C02371=1084,32291,-28357,1060,-27667,-1162
C02372=1082,32304,-28341,1060,-27672,-1161
C02373=1120,32308,-28336,1055,-27674,-1176
C02374=1156,32305,-28339,1050,-27673,-1190
C02375=1195,32311,-28332,1044,-27676,-1205
C02376=1230,32306,-28337,1039,-27674,-1219
C02377=1269,32312,-28330,1034,-27677,-1234
C02378=1304,32324,-28315,1028,-27682,-1248
C02379=1341,32332,-28305,1023,-27685,-1262
C02380=1378,32340,-28295,1018,-27689,-1277
C02381=1414,32352,-28280,1012,-27693,-1290
C02382=1452,32358,-28273,1007,-27696,-1305
C02383=1486,32373,-28255,1002,-27702,-1318
C02384=1521,32386,-28239,997,-27707,-1332
C02385=1556,32397,-28225,992,-27712,-1345
C02386=1592,32409,-28211,986,-27716,-1359
C02387=1624,32426,-28189,982,-27723,-1372
C02388=1655,32445,-28166,977,-27730,-1384
C02389=1688,32462,-28146,972,-27737,-1396
C02390=1718,32483,-28120,968,-27745,-1408
C02391=1749,32503,-28095,963,-27753,-1420
C02392=1781,32521,-28074,958,-27760,-1432
C02393=1810,32545,-28045,954,-27769,-1443
C02394=1838,32569,-28015,950,-27778,-1454
C02395=1867,32592,-27986,945,-27787,-1465
C02396=1892,32623,-27950,941,-27799,-1475
C02397=1921,32646,-27921,937,-27808,-1486
C02398=1946,32677,-27884,933,-27819,-1495
C02399=1971,32707,-27847,929,-27831,-1505
C02400=1996,32737,-27811,925,-27842,-1514
C02401=2022,32766,-27775,921,-27853,-1524
C02402=2018,32742,-27804,922,-27844,-1523
C02403=1993,32712,-27841,926,-27833,-1513
C02404=1975,32680,-27879,929,-27821,-1507
C02405=1950,32651,-27915,933,-27809,-1497
C02406=1921,32626,-27945,937,-27800,-1486
C02407=1896,32596,-27982,941,-27789,-1476
C02408=1867,32572,-28011,945,-27780,-1465
C02409=1839,32548,-28040,950,-27770,-1454
C02410=1810,32524,-28069,954,-27761,-1443
C02411=1781,32501,-28098,958,-27752,-1432
C02412=1752,32478,-28125,963,-27744,-1421
C02413=1718,32464,-28143,968,-27738,-1408
C02414=1688,32441,-28170,972,-27729,-1397
C02415=1655,32426,-28189,977,-27723,-1384
C02416=1621,32411,-28207,982,-27717,-1371
C02417=1589,32395,-28227,987,-27711,-1358
C02418=1554,32382,-28243,992,-27706,-1345
C02419=1520,32368,-28260,997,-27700,-1331
C02420=1486,32353,-28278,1002,-27695,-1318
C02421=1450,32343,-28291,1007,-27690,-1304
C02422=1413,32333,-28303,1013,-27686,-1290
C02423=1375,32328,-28310,1018,-27684,-1275
C02424=1341,32313,-28328,1023,-27678,-1262
C02425=1304,32304,-28340,1029,-27674,-1248
C02426=1268,32293,-28353,1034,-27670,-1234
C02427=1268,32293,-26953,1034,-27670,-1234
C02428=1269,32446,-24168,1032,-27726,-1233
C02429=1269,32446,-28168,1032,-27726,-1233
C02430=1230,32450,-28164,1037,-27727,-1218
C02431=1188,32444,-28172,1043,-27724,-1201
C02432=1149,32447,-28167,1049,-27726,-1186
C02433=1111,32451,-28163,1054,-27727,-1171
C02434=1072,32455,-28159,1060,-27728,-1156
C02435=1033,32459,-28154,1065,-27729,-1141
C02436=998,32473,-28138,1070,-27733,-1127
C02437=960,32477,-28133,1075,-27734,-1112
C02438=925,32491,-28117,1080,-27739,-1098
C02439=889,32503,-28103,1085,-27743,-1084
C02440=855,32519,-28084,1090,-27749,-1071
C02441=819,32530,-28070,1095,-27752,-1056
C02442=785,32547,-28050,1099,-27758,-1043
C02443=753,32571,-28022,1104,-27767,-1030
C02444=719,32589,-28001,1108,-27773,-1017
C02445=688,32613,-27972,1112,-27781,-1005
C02446=660,32639,-27940,1116,-27791,-994
C02447=632,32665,-27909,1119,-27800,-982
C02448=608,32693,-27876,1123,-27810,-973
C02449=590,32725,-26437,1125,-27821,-965
C02450=-41004,59868,4099,4900,-34257,16705
C02451=-41004,59868,1099,4900,-34257,16705
C02452=-41004,64596,1380,5213,-31659,16463
C02453=-41004,59868,1099,4900,-34257,16705
C02454=-41004,59868,9099,4900,-34257,16705
C02455=590,32725,-23837,1125,-27821,-965
C02456=590,32725,-27837,1125,-27821,-965
C02457=565,32753,-27804,1128,-27831,-955
C02458=553,32788,-27762,1129,-27844,-950
C02459=541,32823,-27720,1130,-27857,-945
C02460=540,32836,-27704,1130,-27862,-945
C02461=558,32804,-27742,1128,-27850,-952
C02462=576,32772,-27781,1126,-27839,-959
C02463=600,32744,-27814,1123,-27828,-969
C02464=618,32712,-27853,1121,-27817,-976
C02465=642,32684,-27886,1118,-27807,-986
C02466=674,32660,-27915,1114,-27798,-999
C02467=698,32632,-27949,1110,-27788,-1009
C02468=730,32608,-27978,1106,-27780,-1021
C02469=761,32583,-28007,1102,-27771,-1034
C02470=795,32566,-28027,1098,-27765,-1047
C02471=829,32549,-28047,1093,-27759,-1060
C02472=863,32532,-28068,1088,-27753,-1074
C02473=897,32516,-28087,1084,-27748,-1087
C02474=933,32505,-28100,1079,-27744,-1101
C02475=970,32495,-28112,1074,-27741,-1116
C02476=1006,32485,-28123,1069,-27738,-1130
C02477=1044,32480,-28129,1063,-27736,-1145
C02478=1082,32472,-28138,1058,-27734,-1160
C02479=1121,32469,-28141,1053,-27733,-1175
C02480=1159,32466,-28145,1047,-27733,-1190
C02481=1199,32464,-28147,1042,-27732,-1205
C02482=1240,32468,-28142,1036,-27734,-1221
C02483=1279,32466,-28143,1030,-27734,-1237
C02484=1321,32473,-28136,1024,-27737,-1253
C02485=1364,32479,-28128,1018,-27739,-1270
C02486=1401,32494,-28109,1013,-27745,-1284
C02487=1443,32500,-28102,1007,-27748,-1300
C02488=1478,32520,-28077,1001,-27756,-1314
C02489=1512,32537,-28056,996,-27763,-1327
C02490=1502,32518,-28079,998,-27755,-1323
C02491=1469,32494,-28108,1003,-27746,-1311
C02492=1432,32479,-28127,1008,-27740,-1296
C02493=1390,32473,-28134,1014,-27738,-1280
C02494=1351,32461,-28149,1020,-27733,-1265
C02495=1311,32452,-28161,1026,-27729,-1249
C02496=1269,32446,-28168,1032,-27726,-1233
C02497=1269,32446,-26768,1032,-27726,-1233
C02498=1271,32618,-23960,1029,-27790,-1232
C02499=1271,32618,-27960,1029,-27790,-1232
C02500=1216,32620,-27959,1037,-27790,-1211
C02501=1161,32621,-27958,1045,-27790,-1190
C02502=1110,32633,-27944,1052,-27793,-1169
C02503=1059,32644,-27930,1059,-27797,-1149
C02504=1009,32662,-27909,1066,-27803,-1130
C02505=963,32688,-27879,1072,-27812,-1111
C02506=915,32709,-27853,1079,-27819,-1092
C02507=871,32742,-27814,1085,-27831,-1075
C02508=827,32776,-27774,1090,-27843,-1058
C02509=790,32813,-27729,1095,-27856,-1043
C02510=756,32852,-27682,1099,-27870,-1029
C02511=724,32892,-27634,1103,-27885,-1016
C02512=700,32937,-27580,1106,-27901,-1007
C02513=670,32978,-27531,1110,-27916,-995
C02514=660,33023,-27477,1111,-27932,-990
C02515=689,32981,-27527,1107,-27917,-1002
C02516=719,32940,-27576,1103,-27902,-1014
C02517=749,32899,-27626,1100,-27887,-1026
C02518=785,32861,-27672,1095,-27874,-1040
C02519=816,32820,-27720,1091,-27859,-1053
C02520=853,32783,-27765,1087,-27846,-1068
C02521=897,32749,-27806,1081,-27834,-1085
C02522=943,32722,-27837,1075,-27825,-1103
C02523=989,32696,-27869,1069,-27815,-1122
C02524=1038,32676,-27892,1062,-27809,-1141
C02525=1087,32658,-27914,1055,-27802,-1160
C02526=1138,32646,-27927,1048,-27799,-1180
C02527=1193,32645,-27929,1040,-27799,-1202
C02528=1248,32643,-27930,1032,-27799,-1223
C02529=1303,32642,-27931,1025,-27799,-1245
C02530=1361,32650,-27920,1016,-27803,-1267
C02531=1420,32659,-27910,1008,-27807,-1290
C02532=1478,32668,-27899,1000,-27810,-1313
C02533=1532,32685,-27877,992,-27817,-1333
C02534=1586,32700,-27858,984,-27824,-1355
C02535=1639,32720,-27834,976,-27832,-1375
C02536=1692,32737,-27813,968,-27839,-1396
C02537=1741,32763,-27781,961,-27849,-1415
C02538=1789,32790,-27749,954,-27859,-1433
C02539=1838,32816,-27716,947,-27869,-1452
C02540=1879,32856,-27668,941,-27885,-1468
C02541=1921,32895,-27620,934,-27900,-1484
C02542=1962,32934,-27572,928,-27915,-1500
C02543=2000,32980,-27517,922,-27932,-1514
C02544=2009,32970,-27529,921,-27928,-1518
C02545=1978,32923,-27586,926,-27910,-1506
C02546=1939,32878,-27640,932,-27894,-1491
C02547=1899,32838,-27690,938,-27878,-1476
C02548=1857,32798,-27738,944,-27863,-1460
C02549=1809,32771,-27771,951,-27853,-1441
C02550=1759,32747,-27801,959,-27843,-1422
C02551=1711,32721,-27833,966,-27833,-1403
C02552=1661,32697,-27862,973,-27823,-1384
C02553=1608,32677,-27886,981,-27815,-1364
C02554=1554,32662,-27905,989,-27809,-1342
C02555=1496,32651,-27919,997,-27805,-1320
C02556=1438,32643,-27929,1006,-27801,-1297
C02557=1385,32625,-27951,1013,-27794,-1277
C02558=1326,32617,-27962,1022,-27790,-1254
C02559=1271,32618,-27960,1029,-27790,-1232
C02560=1271,32618,-26560,1029,-27790,-1232
C02561=998,32374,-24257,1071,-27697,-1128
C02562=998,32374,-28257,1071,-27697,-1128
C02563=1004,32369,-28263,1071,-27695,-1130
C02564=994,32367,-28265,1072,-27694,-1126
C02565=985,32366,-28267,1073,-27694,-1123
C02566=975,32365,-28269,1075,-27693,-1119
C02567=965,32363,-28271,1076,-27692,-1115
C02568=958,32369,-28264,1077,-27694,-1112
C02569=950,32371,-28262,1078,-27695,-1109
C02570=940,32369,-28264,1080,-27694,-1105
C02571=932,32371,-28261,1081,-27695,-1102
C02572=924,32376,-28255,1082,-27697,-1099
C02573=915,32375,-28257,1083,-27696,-1095
C02574=908,32381,-28250,1084,-27698,-1092
C02575=899,32382,-28248,1085,-27699,-1089
C02576=891,32385,-28245,1086,-27699,-1086
C02577=883,32389,-28240,1087,-27701,-1083
C02578=874,32389,-28241,1089,-27701,-1079
C02579=867,32394,-28234,1090,-27703,-1076
C02580=858,32395,-28233,1091,-27703,-1073
C02581=850,32398,-28230,1092,-27704,-1070
C02582=842,32403,-28224,1093,-27705,-1067
C02583=833,32402,-28225,1094,-27705,-1063
C02584=826,32408,-28218,1095,-27707,-1060
C02585=817,32408,-28217,1097,-27707,-1057
C02586=809,32411,-28214,1098,-27708,-1054
C02587=801,32416,-28209,1099,-27710,-1051
C02588=792,32415,-28209,1100,-27710,-1047
C02589=785,32421,-28202,1101,-27712,-1044
C02590=777,32427,-28196,1102,-27714,-1041
C02591=770,32432,-28189,1103,-27716,-1038
C02592=763,32438,-28183,1104,-27718,-1036
C02593=761,32446,-28172,1104,-27721,-1035
C02594=767,32444,-28175,1103,-27720,-1037
C02595=775,32440,-28179,1102,-27719,-1040
C02596=784,32440,-28180,1101,-27718,-1044
C02597=791,32434,-28187,1100,-27717,-1047
C02598=798,32429,-28193,1099,-27715,-1049
C02599=806,32426,-28196,1098,-27714,-1053
C02600=815,32425,-28198,1097,-27713,-1056
C02601=822,32419,-28204,1096,-27711,-1059
C02602=832,32420,-28203,1094,-27712,-1063
C02603=839,32415,-28209,1093,-27710,-1065
C02604=848,32413,-28212,1092,-27709,-1069
C02605=856,32411,-28214,1091,-27709,-1072
C02606=863,32406,-28220,1090,-27707,-1075
C02607=870,32400,-28227,1089,-27705,-1078
C02608=879,32398,-28229,1088,-27704,-1081
C02609=889,32400,-28227,1087,-27705,-1085
C02610=897,32398,-28230,1085,-27704,-1088
C02611=904,32393,-28236,1084,-27702,-1091
C02612=914,32394,-28234,1083,-27703,-1095
C02613=921,32388,-28241,1082,-27701,-1098
C02614=930,32387,-28243,1081,-27701,-1101
C02615=938,32384,-28245,1080,-27700,-1104
C02616=945,32379,-28251,1079,-27698,-1107
C02617=955,32381,-28249,1077,-27699,-1111
C02618=965,32382,-28248,1076,-27699,-1115
C02619=972,32376,-28255,1075,-27697,-1118
C02620=980,32375,-28256,1074,-27697,-1121
C02621=990,32376,-28255,1072,-27698,-1125
C02622=998,32374,-26857,1071,-27697,-1128
C02623=-41004,59868,4099,4900,-34257,16705
C02624=-41004,59868,1099,4900,-34257,16705
C02625=-41004,64596,1380,5213,-31659,16463
C02626=-41004,59868,1099,4900,-34257,16705
C02627=-41004,59868,9099,4900,-34257,16705
C02628=998,32374,-24257,1071,-27697,-1128
C02629=998,32374,-28257,1071,-27697,-1128
C02630=998,32374,-26857,1071,-27697,-1128
C02631=975,32976,-23531,1067,-27918,-1114
C02632=975,32976,-27531,1067,-27918,-1114
C02633=961,32984,-27522,1069,-27921,-1108
C02634=947,32989,-27515,1071,-27923,-1103
C02635=934,32999,-27503,1072,-27926,-1097
C02636=921,33009,-27491,1074,-27930,-1092
C02637=913,33022,-27476,1075,-27935,-1089
C02638=902,33033,-27463,1077,-27939,-1085
C02639=889,33043,-27451,1078,-27942,-1079
C02640=881,33056,-27435,1079,-27947,-1076
C02641=871,33067,-27422,1081,-27951,-1072
C02642=864,33080,-27406,1081,-27956,-1069
C02643=857,33094,-27389,1082,-27961,-1067
C02644=848,33106,-27374,1083,-27965,-1063
C02645=838,33118,-27361,1084,-27969,-1059
C02646=832,33132,-27344,1085,-27974,-1056
C02647=826,33146,-27327,1086,-27979,-1054
C02648=816,33157,-27314,1087,-27983,-1050
C02649=807,33169,-27299,1088,-27988,-1046
C02650=804,33185,-27280,1088,-27994,-1045
C02651=795,33197,-27266,1090,-27998,-1041
C02652=793,33213,-27246,1090,-28004,-1040
C02653=789,33228,-27228,1090,-28009,-1039
C02654=781,33241,-27213,1091,-28014,-1036
C02655=780,33258,-27192,1091,-28020,-1035
C02656=779,33275,-27172,1091,-28026,-1034
C02657=771,33287,-27157,1092,-28031,-1031
C02658=767,33303,-27139,1092,-28036,-1030
C02659=766,33319,-27118,1092,-28042,-1029
C02660=765,33336,-27098,1092,-28049,-1029
C02661=764,33353,-27078,1092,-28055,-1028
C02662=766,33363,-27066,1091,-28059,-1029
C02663=774,33350,-27081,1090,-28054,-1032
C02664=775,33333,-27101,1091,-28048,-1032
C02665=776,33317,-27121,1091,-28042,-1033
C02666=784,33304,-27137,1090,-28037,-1036
C02667=788,33289,-27155,1089,-28032,-1038
C02668=789,33272,-27175,1089,-28025,-1038
C02669=790,33255,-27195,1089,-28019,-1039
C02670=800,33244,-27209,1088,-28015,-1043
C02671=802,33227,-27229,1088,-28009,-1044
C02672=808,33214,-27245,1088,-28004,-1046
C02673=813,33199,-27263,1087,-27999,-1048
C02674=820,33186,-27279,1086,-27994,-1051
C02675=825,33171,-27296,1086,-27989,-1053
C02676=833,33158,-27312,1085,-27984,-1056
C02677=839,33145,-27328,1084,-27979,-1059
C02678=847,33132,-27344,1083,-27974,-1062
C02679=857,33121,-27357,1082,-27970,-1066
C02680=864,33107,-27374,1081,-27965,-1069
C02681=870,33093,-27390,1080,-27960,-1072
C02682=880,33081,-27405,1079,-27956,-1075
C02683=889,33069,-27419,1078,-27952,-1079
C02684=901,33059,-27432,1076,-27948,-1084
C02685=908,33046,-27447,1075,-27943,-1087
C02686=921,33036,-27459,1074,-27940,-1092
C02687=933,33025,-27472,1072,-27936,-1097
C02688=940,33012,-27488,1071,-27931,-1100
C02689=953,33002,-27500,1070,-27928,-1105
C02690=966,32992,-27512,1068,-27924,-1110
C02691=979,32982,-27524,1066,-27921,-1115
C02692=975,32976,-27531,1067,-27918,-1114
C02693=975,32976,-26131,1067,-27918,-1114
C02694=1115,33029,-23465,1046,-27940,-1168
C02695=1115,33029,-27465,1046,-27940,-1168
C02696=1109,33039,-27453,1047,-27943,-1166
C02697=1102,33049,-27442,1048,-27947,-1163
C02698=1092,33057,-27432,1050,-27950,-1159
C02699=1087,33068,-27419,1050,-27954,-1157
C02700=1078,33076,-27409,1051,-27957,-1153
C02701=1074,33088,-27395,1052,-27961,-1152
C02702=1066,33097,-27384,1053,-27964,-1148
C02703=1061,33108,-27371,1053,-27968,-1146
C02704=1054,33118,-27359,1054,-27972,-1144
C02705=1047,33127,-27348,1055,-27975,-1140
C02706=1043,33139,-27334,1055,-27979,-1139
C02707=1033,33147,-27324,1057,-27982,-1135
C02708=1032,33160,-27308,1057,-27987,-1134
C02709=1026,33170,-27296,1057,-27991,-1132
C02710=1021,33181,-27283,1058,-27995,-1130
C02711=1029,33177,-27288,1057,-27993,-1133
C02712=1039,33169,-27297,1056,-27990,-1137
C02713=1043,33157,-27311,1055,-27986,-1139
C02714=1052,33149,-27321,1054,-27983,-1142
C02715=1056,33138,-27335,1053,-27979,-1144
C02716=1064,33128,-27346,1053,-27976,-1147
C02717=1070,33118,-27358,1052,-27972,-1150
C02718=1075,33107,-27371,1051,-27968,-1152
C02719=1084,33099,-27382,1050,-27965,-1155
C02720=1087,33087,-27396,1050,-27961,-1157
C02721=1097,33079,-27406,1049,-27958,-1160
C02722=1101,33067,-27419,1048,-27954,-1162
C02723=1111,33059,-27429,1047,-27951,-1166
C02724=1121,33052,-27438,1045,-27948,-1170
C02725=1132,33044,-27448,1044,-27945,-1174
C02726=1142,33036,-27457,1043,-27943,-1178
C02727=1152,33028,-27467,1041,-27940,-1182
C02728=1163,33023,-27473,1040,-27938,-1187
C02729=1175,33019,-27477,1038,-27937,-1191
C02730=1187,33017,-27480,1037,-27936,-1196
C02731=1198,33010,-27487,1035,-27934,-1201
C02732=1211,33010,-27488,1033,-27934,-1205
C02733=1221,33003,-27496,1032,-27931,-1210
C02734=1235,33005,-27494,1030,-27932,-1215
C02735=1246,33000,-27499,1028,-27931,-1219
C02736=1259,32999,-27501,1027,-27930,-1224
C02737=1272,32999,-27501,1025,-27930,-1229
C02738=1282,32992,-27508,1023,-27928,-1234
C02739=1294,32990,-27511,1022,-27927,-1238
C02740=1294,32985,-27517,1022,-27925,-1238
C02741=1281,32983,-27520,1024,-27925,-1233
C02742=1270,32991,-27511,1025,-27927,-1229
C02743=1257,32989,-27513,1027,-27926,-1224
C02744=1245,32992,-27509,1029,-27928,-1219
C02745=1233,32995,-27506,1030,-27928,-1214
C02746=1220,32994,-27507,1032,-27928,-1209
C02747=1209,33001,-27499,1034,-27930,-1205
C02748=1196,32999,-27501,1036,-27930,-1200
C02749=1184,33003,-27496,1037,-27931,-1195
C02750=1172,33005,-27494,1039,-27931,-1190
C02751=1161,33012,-27486,1040,-27934,-1186
C02752=1149,33013,-27485,1042,-27934,-1181
C02753=1138,33019,-27477,1043,-27936,-1177
C02754=1126,33021,-27475,1045,-27937,-1172
C02755=1115,33029,-27465,1046,-27940,-1168
C02756=1115,33029,-26065,1046,-27940,-1168
C02757=1159,33118,-23358,1039,-27973,-1185
C02758=1159,33118,-27358,1039,-27973,-1185
C02759=1098,33196,-27264,1047,-28001,-1160
C02760=1121,33177,-27286,1044,-27995,-1169
C02761=1204,33114,-27363,1033,-27972,-1202
C02762=1299,33071,-27413,1020,-27957,-1239
C02763=1397,33036,-27454,1007,-27946,-1278
C02764=1499,33015,-27479,992,-27939,-1318
C02765=1611,33022,-27470,977,-27943,-1362
C02766=1719,33039,-27448,961,-27951,-1404
C02767=1667,33068,-27414,968,-27961,-1383
C02768=1559,33073,-27408,983,-27961,-1341
C02769=1460,33104,-27371,997,-27972,-1302
C02770=1365,33150,-27317,1010,-27987,-1265
C02771=1278,33217,-27237,1021,-28011,-1230
C02772=1200,33289,-27151,1031,-28037,-1199
C02773=1136,33369,-27055,1039,-28065,-1173
C02774=1085,33456,-26950,1045,-28097,-1153
C02775=1055,33555,-26831,1049,-28133,-1140
C02776=1038,33661,-26703,1050,-28172,-1132
C02777=1048,33768,-26573,1047,-28212,-1136
C02778=1081,33870,-26451,1041,-28250,-1148
C02779=1142,33964,-26336,1031,-28285,-1171
C02780=1176,33974,-26324,1027,-28289,-1184
C02781=1101,33883,-26435,1038,-28255,-1155
C02782=1069,33781,-26558,1044,-28217,-1144
C02783=1066,33672,-26690,1045,-28176,-1144
C02784=1083,33565,-26818,1044,-28137,-1151
C02785=1110,33465,-26940,1042,-28100,-1162
C02786=1162,33378,-27043,1036,-28069,-1184
C02787=1229,33300,-27137,1027,-28041,-1210
C02788=1303,33226,-27226,1018,-28015,-1240
C02789=1392,33166,-27298,1006,-27993,-1275
C02790=1485,33118,-27355,993,-27977,-1312
C02791=1585,33088,-27390,979,-27967,-1351
C02792=1693,33081,-27397,964,-27966,-1393
C02793=1800,33112,-27359,949,-27978,-1435
C02794=1758,33139,-27327,955,-27988,-1418
C02795=1697,33139,-27327,963,-27987,-1395
C02796=1631,33177,-27282,972,-28001,-1368
C02797=1529,33201,-27254,986,-28008,-1328
C02798=1435,33248,-25798,999,-28024,-1291
C02799=-41004,59868,4099,4900,-34257,16705
C02800=-41004,59868,1099,4900,-34257,16705
C02801=-41004,64596,1380,5213,-31659,16463
C02802=-41004,59868,1099,4900,-34257,16705
C02803=-41004,59868,9099,4900,-34257,16705
C02804=1435,33248,-23198,999,-28024,-1291
C02805=1435,33248,-27198,999,-28024,-1291
C02806=1355,33319,-27113,1009,-28050,-1259
C02807=1282,33393,-27024,1019,-28076,-1230
C02808=1235,33483,-26916,1024,-28109,-1211
C02809=1200,33579,-26800,1028,-28144,-1197
C02810=1245,33495,-26902,1023,-28113,-1215
C02811=1297,33408,-27006,1016,-28082,-1236
C02812=1370,33334,-27095,1007,-28055,-1265
C02813=1451,33263,-27180,996,-28030,-1297
C02814=1543,33212,-27240,984,-28012,-1334
C02815=1644,33186,-27271,970,-28004,-1373
C02816=1748,33169,-27291,956,-27999,-1414
C02817=1861,33185,-27270,939,-28006,-1458
C02818=1858,33129,-27338,941,-27985,-1457
C02819=1769,33063,-27418,954,-27960,-1423
C02820=1667,33020,-27471,969,-27943,-1384
C02821=1557,32994,-27503,985,-27932,-1341
C02822=1448,32998,-27500,1000,-27932,-1298
C02823=1349,33029,-27464,1014,-27942,-1259
C02824=1252,33067,-27418,1027,-27956,-1221
C02825=1159,33118,-27358,1039,-27973,-1185
C02826=1159,33118,-25958,1039,-27973,-1185
C02827=964,33299,-23141,1064,-28038,-1107
C02828=964,33299,-27141,1064,-28038,-1107
C02829=953,33311,-27126,1066,-28042,-1102
C02830=943,33324,-27111,1067,-28046,-1098
C02831=936,33338,-27094,1068,-28052,-1095
C02832=930,33353,-27076,1069,-28057,-1093
C02833=920,33366,-27061,1070,-28062,-1089
C02834=916,33381,-27042,1070,-28067,-1087
C02835=908,33396,-27025,1071,-28072,-1084
C02836=907,33413,-27004,1071,-28079,-1083
C02837=906,33431,-26983,1071,-28085,-1083
C02838=905,33448,-26961,1071,-28092,-1082
C02839=895,33461,-26946,1072,-28096,-1078
C02840=893,33478,-26925,1072,-28103,-1077
C02841=892,33496,-26904,1072,-28109,-1077
C02842=891,33513,-26883,1072,-28116,-1076
C02843=890,33531,-26862,1072,-28122,-1076
C02844=889,33548,-26841,1072,-28129,-1075
C02845=888,33566,-26819,1072,-28135,-1074
C02846=887,33584,-26798,1072,-28141,-1074
C02847=885,33601,-26777,1072,-28148,-1073
C02848=884,33619,-26756,1072,-28154,-1073
C02849=887,33635,-26736,1071,-28161,-1074
C02850=892,33651,-26716,1070,-28167,-1075
C02851=891,33669,-26695,1070,-28173,-1075
C02852=890,33687,-26674,1070,-28179,-1074
C02853=892,33703,-26654,1069,-28186,-1075
C02854=897,33719,-26634,1069,-28192,-1077
C02855=896,33737,-26613,1069,-28198,-1076
C02856=900,33753,-26593,1068,-28204,-1078
C02857=904,33769,-26574,1067,-28210,-1079
C02858=913,33779,-26562,1066,-28214,-1082
C02859=923,33767,-26577,1064,-28210,-1087
C02860=915,33751,-26595,1066,-28204,-1084
C02861=916,33734,-26616,1066,-28197,-1084
C02862=913,33718,-26636,1066,-28191,-1083
C02863=908,33701,-26656,1067,-28185,-1081
C02864=909,33684,-26677,1067,-28179,-1082
C02865=910,33666,-26698,1067,-28172,-1083
C02866=912,33649,-26719,1067,-28166,-1083
C02867=909,33632,-26740,1068,-28160,-1082
C02868=904,33616,-26759,1069,-28154,-1080
C02869=905,33598,-26780,1069,-28147,-1081
C02870=906,33581,-26801,1069,-28141,-1082
C02871=907,33563,-26822,1069,-28134,-1082
C02872=909,33546,-26844,1069,-28128,-1083
C02873=910,33528,-26865,1069,-28121,-1083
C02874=911,33511,-26886,1069,-28115,-1084
C02875=912,33493,-26907,1069,-28108,-1085
C02876=913,33475,-26928,1069,-28102,-1085
C02877=914,33458,-26950,1069,-28095,-1086
C02878=915,33440,-26971,1070,-28089,-1086
C02879=926,33428,-26986,1068,-28085,-1090
C02880=927,33410,-27007,1068,-28078,-1091
C02881=928,33393,-27028,1068,-28072,-1092
C02882=939,33381,-27043,1067,-28067,-1096
C02883=940,33363,-27064,1067,-28061,-1097
C02884=951,33351,-27079,1066,-28056,-1101
C02885=953,33334,-27099,1066,-28050,-1102
C02886=962,33321,-27114,1064,-28046,-1106
C02887=973,33309,-27129,1063,-28041,-1110
C02888=964,33299,-27141,1064,-28038,-1107
C02889=964,33299,-25741,1064,-28038,-1107
C02890=523,33294,-23151,1127,-28030,-934
C02891=523,33294,-27151,1127,-28030,-934
C02892=524,33274,-27175,1127,-28023,-935
C02893=525,33254,-27200,1127,-28015,-935
C02894=526,33233,-27224,1127,-28008,-936
C02895=536,33218,-27243,1126,-28002,-940
C02896=538,33198,-27267,1126,-27995,-941
C02897=539,33178,-27291,1126,-27988,-942
C02898=541,33158,-27316,1126,-27980,-942
C02899=545,33139,-27338,1125,-27973,-944
C02900=553,33122,-27358,1125,-27967,-947
C02901=554,33102,-27382,1125,-27960,-948
C02902=564,33087,-27400,1123,-27955,-952
C02903=567,33068,-27424,1123,-27947,-953
C02904=576,33052,-27443,1122,-27942,-957
C02905=585,33036,-27462,1121,-27936,-961
C02906=588,33017,-27485,1121,-27929,-962
C02907=599,33002,-27503,1120,-27923,-966
C02908=610,32987,-27521,1118,-27918,-971
C02909=611,32967,-27545,1118,-27911,-971
C02910=622,32952,-27563,1117,-27905,-976
C02911=632,32936,-27582,1116,-27900,-980
C02912=613,32933,-27587,1119,-27898,-973
C02913=611,32952,-27563,1119,-27905,-972
C02914=601,32968,-27544,1120,-27911,-968
C02915=590,32983,-27526,1121,-27916,-963
C02916=584,33000,-27505,1122,-27923,-961
C02917=575,33016,-27486,1123,-27928,-957
C02918=568,33033,-27466,1124,-27935,-954
C02919=557,33048,-27448,1125,-27940,-950
C02920=555,33068,-27424,1125,-27947,-949
C02921=545,33083,-27406,1126,-27953,-945
C02922=538,33100,-27386,1127,-27959,-942
C02923=533,33118,-27363,1127,-27966,-940
C02924=532,33138,-27339,1127,-27973,-939
C02925=524,33155,-27319,1128,-27979,-936
C02926=520,33174,-27296,1129,-27986,-934
C02927=519,33194,-27272,1128,-27993,-933
C02928=518,33214,-27248,1128,-28001,-933
C02929=516,33235,-27223,1128,-28008,-932
C02930=507,33250,-27204,1129,-28014,-928
C02931=505,33270,-27181,1129,-28021,-927
C02932=503,33290,-27156,1129,-28028,-926
C02933=502,33310,-27132,1129,-28036,-926
C02934=501,33331,-27107,1129,-28043,-925
C02935=510,33348,-27086,1128,-28050,-928
C02936=509,33369,-27061,1128,-28058,-928
C02937=507,33389,-27037,1127,-28065,-927
C02938=506,33409,-27012,1127,-28072,-926
C02939=510,33428,-26989,1127,-28080,-928
C02940=514,33447,-26966,1126,-28087,-929
C02941=513,33468,-26942,1126,-28094,-928
C02942=527,33469,-26940,1124,-28095,-934
C02943=523,33454,-26958,1124,-28089,-933
C02944=524,33434,-26983,1124,-28082,-933
C02945=525,33413,-27007,1125,-28074,-934
C02946=524,33394,-27031,1125,-28067,-933
C02947=518,33375,-27053,1126,-28060,-931
C02948=519,33355,-27078,1126,-28053,-932
C02949=520,33335,-27102,1126,-28045,-933
C02950=522,33315,-27126,1126,-28038,-933
C02951=523,33294,-27151,1127,-28030,-934
C02952=523,33294,-25751,1127,-28030,-934
C02953=303,33334,-23105,1157,-28042,-848
C02954=303,33334,-27105,1157,-28042,-848
C02955=303,33367,-27065,1156,-28054,-847
C02956=311,33398,-27027,1155,-28066,-850
C02957=309,33432,-26987,1155,-28078,-849
C02958=317,33463,-26949,1153,-28090,-852
C02959=325,33494,-26911,1152,-28101,-855
C02960=333,33525,-26874,1150,-28113,-858
C02961=341,33557,-26836,1148,-28125,-861
C02962=349,33588,-26799,1147,-28136,-863
C02963=363,33617,-26763,1145,-28147,-868
C02964=379,33647,-26727,1142,-28158,-874
C02965=395,33676,-26692,1139,-28169,-880
C02966=418,33703,-26659,1136,-28180,-889
C02967=433,33732,-26623,1133,-28190,-895
C02968=460,33753,-26598,1129,-28199,-905
C02969=482,33781,-26564,1126,-28209,-914
C02970=508,33802,-26539,1122,-28217,-924
C02971=536,33819,-26517,1118,-28224,-935
C02972=561,33842,-26490,1114,-28233,-944
C02973=591,33856,-26473,1110,-28238,-956
C02974=601,33880,-25043,1108,-28247,-959
C02975=-41004,59868,4099,4900,-34257,16705
C02976=-41004,59868,1099,4900,-34257,16705
C02977=-41004,64596,1380,5213,-31659,16463
C02978=-41004,59868,1099,4900,-34257,16705
C02979=-41004,59868,9099,4900,-34257,16705
C02980=601,33880,-22443,1108,-28247,-959
C02981=601,33880,-26443,1108,-28247,-959
C02982=573,33893,-26427,1112,-28252,-948
C02983=545,33906,-26412,1115,-28256,-937
C02984=517,33920,-26396,1119,-28261,-926
C02985=491,33940,-26372,1122,-28268,-916
C02986=463,33953,-26357,1126,-28272,-905
C02987=438,33973,-26333,1129,-28279,-895
C02988=410,33986,-26317,1133,-28284,-883
C02989=384,34006,-26293,1136,-28291,-873
C02990=359,34027,-26269,1140,-28298,-863
C02991=333,34047,-26245,1143,-28305,-853
C02992=314,34071,-26216,1145,-28314,-845
C02993=292,34093,-26190,1148,-28321,-836
C02994=271,34116,-26162,1151,-28330,-828
C02995=251,34139,-26134,1153,-28338,-820
C02996=232,34131,-26144,1156,-28335,-812
C02997=233,34098,-26184,1156,-28322,-813
C02998=245,34070,-26218,1155,-28312,-818
C02999=247,34036,-26259,1155,-28300,-819
C03000=248,34002,-26299,1155,-28287,-820
C03001=250,33969,-26340,1156,-28275,-821
C03002=252,33935,-26381,1156,-28263,-822
C03003=254,33901,-26421,1156,-28250,-823
C03004=256,33868,-26462,1156,-28238,-824
C03005=258,33834,-26502,1156,-28226,-825
C03006=260,33800,-26543,1157,-28213,-826
C03007=261,33767,-26583,1157,-28201,-827
C03008=263,33733,-26624,1157,-28189,-828
C03009=265,33699,-26665,1157,-28176,-829
C03010=267,33666,-26705,1157,-28164,-830
C03011=269,33632,-26746,1158,-28152,-832
C03012=271,33599,-26786,1158,-28139,-833
C03013=273,33565,-26827,1158,-28127,-834
C03014=275,33531,-26867,1158,-28114,-835
C03015=276,33498,-26908,1158,-28102,-836
C03016=270,33466,-26946,1160,-28090,-833
C03017=270,33433,-26986,1160,-28078,-834
C03018=272,33399,-27027,1160,-28066,-835
C03019=274,33366,-27067,1160,-28053,-836
C03020=276,33332,-27108,1161,-28041,-837
C03021=303,33334,-27105,1157,-28042,-848
C03022=303,33334,-25705,1157,-28042,-848
C03023=1429,33520,-22870,996,-28125,-1287
C03024=1429,33520,-26870,996,-28125,-1287
C03025=1428,33538,-26848,996,-28131,-1286
C03026=1417,33551,-26832,998,-28136,-1282
C03027=1416,33569,-26811,998,-28143,-1281
C03028=1407,33583,-26794,999,-28148,-1277
C03029=1404,33600,-26773,999,-28154,-1276
C03030=1403,33618,-26751,999,-28161,-1276
C03031=1401,33636,-26729,999,-28167,-1275
C03032=1400,33655,-26707,999,-28174,-1274
C03033=1402,33667,-26693,999,-28179,-1275
C03034=1410,33652,-26710,998,-28173,-1278
C03035=1411,33634,-26732,998,-28167,-1279
C03036=1418,33619,-26751,997,-28161,-1281
C03037=1423,33603,-26770,996,-28155,-1284
C03038=1425,33585,-26791,996,-28149,-1284
C03039=1433,33571,-26808,995,-28144,-1288
C03040=1437,33554,-26829,995,-28137,-1289
C03041=1447,33541,-26844,994,-28133,-1294
C03042=1449,33523,-26866,994,-28126,-1294
C03043=1457,33508,-26884,993,-28121,-1298
C03044=1461,33492,-26904,992,-28115,-1299
C03045=1472,33479,-26919,991,-28110,-1304
C03046=1479,33464,-26937,990,-28105,-1307
C03047=1484,33448,-26956,990,-28099,-1309
C03048=1494,33435,-26972,988,-28094,-1313
C03049=1502,33420,-26990,987,-28089,-1316
C03050=1509,33405,-27007,987,-28083,-1319
C03051=1517,33391,-27025,986,-28078,-1322
C03052=1528,33378,-27040,984,-28074,-1327
C03053=1538,33365,-27056,983,-28069,-1331
C03054=1546,33350,-27073,982,-28064,-1334
C03055=1553,33336,-27091,981,-28058,-1337
C03056=1568,33325,-27104,979,-28054,-1342
C03057=1575,33310,-27122,978,-28049,-1346
C03058=1589,33299,-27135,976,-28045,-1351
C03059=1603,33288,-27148,975,-28041,-1357
C03060=1611,33274,-27166,974,-28036,-1360
C03061=1625,33263,-27179,972,-28032,-1365
C03062=1639,33252,-27192,970,-28028,-1371
C03063=1637,33245,-27200,970,-28026,-1370
C03064=1621,33252,-27191,973,-28028,-1364
C03065=1606,33260,-27182,975,-28031,-1358
C03066=1591,33271,-27169,976,-28035,-1352
C03067=1577,33282,-27156,978,-28038,-1347
C03068=1570,33296,-27139,979,-28044,-1344
C03069=1556,33307,-27125,981,-28048,-1338
C03070=1548,33322,-27108,982,-28053,-1335
C03071=1534,33333,-27095,984,-28057,-1329
C03072=1526,33348,-27077,985,-28062,-1326
C03073=1512,33358,-27064,987,-28066,-1321
C03074=1505,33373,-27046,988,-28071,-1317
C03075=1497,33388,-27029,988,-28077,-1314
C03076=1487,33401,-27013,990,-28082,-1310
C03077=1482,33417,-26993,990,-28087,-1308
C03078=1475,33432,-26976,991,-28093,-1305
C03079=1464,33445,-26960,992,-28097,-1301
C03080=1453,33458,-26945,994,-28102,-1297
C03081=1452,33476,-26923,994,-28109,-1296
C03082=1441,33489,-26907,995,-28113,-1292
C03083=1437,33505,-26887,995,-28119,-1290
C03084=1429,33520,-26870,996,-28125,-1287
C03085=1429,33520,-25470,996,-28125,-1287
C03086=1682,33546,-22836,961,-28138,-1386
C03087=1682,33546,-26836,961,-28138,-1386
C03088=1695,33511,-26879,959,-28125,-1391
C03089=1708,33475,-26921,958,-28112,-1396
C03090=1729,33445,-26958,955,-28101,-1405
C03091=1751,33415,-26994,952,-28090,-1414
C03092=1774,33384,-27030,950,-28079,-1423
C03093=1796,33354,-27066,947,-28068,-1431
C03094=1821,33326,-27100,944,-28058,-1442
C03095=1855,33306,-27125,939,-28051,-1455
C03096=1890,33291,-27142,934,-28046,-1469
C03097=1924,33274,-27163,930,-28040,-1482
C03098=1961,33263,-27175,924,-28036,-1497
C03099=2000,33260,-27178,919,-28036,-1512
C03100=2039,33256,-27183,914,-28035,-1527
C03101=2076,33271,-27164,908,-28041,-1542
C03102=2115,33268,-27168,903,-28040,-1557
C03103=2144,33292,-27138,898,-28049,-1568
C03104=2111,33315,-27111,903,-28057,-1555
C03105=2072,33319,-27107,908,-28058,-1540
C03106=2033,33322,-27103,914,-28059,-1525
C03107=1997,33334,-27089,919,-28063,-1510
C03108=1962,33350,-27070,923,-28068,-1497
C03109=1928,33369,-27048,928,-28075,-1483
C03110=1901,33396,-27015,932,-28085,-1472
C03111=1877,33425,-26980,935,-28095,-1463
C03112=1856,33456,-26943,937,-28106,-1454
C03113=1834,33486,-26907,940,-28117,-1446
C03114=1814,33518,-26869,942,-28129,-1438
C03115=1800,33552,-26827,944,-28141,-1432
C03116=1787,33588,-26785,945,-28154,-1426
C03117=1775,33623,-26742,947,-28167,-1421
C03118=1771,33664,-26692,947,-28182,-1420
C03119=1759,33699,-26650,948,-28195,-1414
C03120=1756,33740,-26600,948,-28210,-1413
C03121=1762,33779,-26554,947,-28225,-1415
C03122=1769,33817,-26507,945,-28239,-1418
C03123=1781,33854,-26462,943,-28253,-1422
C03124=1794,33891,-26418,941,-28267,-1427
C03125=1819,33925,-26377,937,-28279,-1436
C03126=1844,33954,-26341,933,-28291,-1446
C03127=1877,33978,-26312,929,-28300,-1458
C03128=1913,33994,-26292,923,-28306,-1472
C03129=1934,34020,-26261,920,-28316,-1480
C03130=1900,34037,-26240,925,-28322,-1467
C03131=1863,34048,-26228,930,-28325,-1453
C03132=1827,34058,-26215,935,-28329,-1438
C03133=1795,34047,-26229,939,-28324,-1426
C03134=1761,34027,-26254,944,-28316,-1413
C03135=1731,34000,-26287,949,-28306,-1401
C03136=1703,33967,-26327,953,-28293,-1391
C03137=1683,33931,-26370,956,-28280,-1383
C03138=1675,33893,-26416,958,-28266,-1380
C03139=1664,33856,-26461,960,-28252,-1376
C03140=1652,33819,-26506,962,-28238,-1372
C03141=1651,33779,-26554,962,-28223,-1372
C03142=1648,33740,-26602,963,-28209,-1371
C03143=1651,33699,-26651,963,-28194,-1372
C03144=1655,33658,-26700,963,-28179,-1374
C03145=1667,33623,-26743,962,-28166,-1379
C03146=1670,33582,-26793,962,-28151,-1380
C03147=1682,33546,-25436,961,-28138,-1386
C03148=-41004,59868,4099,4900,-34257,16705
C03149=-41004,59868,1099,4900,-34257,16705
C03150=-41004,64596,1380,5213,-31659,16463
C03151=-41004,59868,1099,4900,-34257,16705
C03152=-41004,59868,9099,4900,-34257,16705
C03153=1682,33546,-22836,961,-28138,-1386
C03154=1682,33546,-26836,961,-28138,-1386
C03155=1682,33546,-25436,961,-28138,-1386
C03156=1856,33512,-22875,937,-28127,-1454
C03157=1856,33512,-26875,937,-28127,-1454
C03158=1974,33377,-27037,921,-28079,-1501
C03159=2151,33340,-27081,897,-28067,-1571
C03160=2340,33372,-27041,870,-28081,-1644
C03161=2512,33450,-26944,845,-28112,-1711
C03162=2684,33529,-26847,820,-28143,-1777
C03163=2856,33605,-26754,795,-28174,-1844
C03164=3022,33693,-26646,770,-28208,-1909
C03165=3169,33814,-26497,749,-28255,-1965
C03166=3326,33900,-26392,726,-28289,-2026
C03167=3484,34001,-26269,703,-28328,-2087
C03168=3644,34095,-26153,679,-28365,-2149
C03169=3479,34101,-26148,703,-28365,-2085
C03170=3332,33982,-26293,724,-28319,-2028
C03171=3201,33903,-26389,743,-28289,-1977
C03172=3344,34029,-26236,722,-28337,-2033
C03173=3484,34160,-26075,701,-28388,-2086
C03174=3612,34311,-25892,682,-28445,-2136
C03175=3723,34470,-25698,665,-28506,-2178
C03176=3825,34622,-25513,650,-28564,-2217
C03177=3689,34665,-25463,669,-28578,-2164
C03178=3555,34527,-25631,689,-28525,-2112
C03179=3420,34389,-25799,709,-28472,-2060
C03180=3274,34270,-25945,730,-28426,-2004
C03181=3121,34161,-26078,752,-28383,-1944
C03182=3199,34325,-25878,740,-28445,-1974
C03183=3331,34470,-25703,720,-28501,-2025
C03184=3462,34614,-25527,701,-28556,-2075
C03185=3576,34767,-25339,684,-28615,-2119
C03186=3671,34931,-25140,669,-28677,-2155
C03187=3638,35070,-24972,673,-28728,-2142
C03188=3490,34958,-25109,694,-28684,-2084
C03189=3352,34827,-25270,714,-28634,-2031
C03190=3218,34689,-25438,734,-28581,-1979
C03191=3086,34545,-25614,754,-28525,-1928
C03192=2957,34394,-25797,773,-28468,-1879
C03193=2973,34446,-25735,771,-28487,-1885
C03194=3100,34598,-25549,751,-28545,-1934
C03195=3232,34742,-25374,732,-28601,-1985
C03196=3368,34878,-25208,712,-28653,-2037
C03197=3478,35008,-25049,695,-28703,-2080
C03198=3306,35030,-25024,719,-28709,-2012
C03199=3156,34922,-25157,741,-28667,-1953
C03200=3005,34814,-25289,763,-28624,-1895
C03201=2869,34676,-25458,783,-28571,-1843
C03202=2735,34535,-25630,803,-28517,-1791
C03203=2834,34674,-25461,788,-28570,-1829
C03204=2966,34818,-25285,768,-28625,-1880
C03205=3117,34926,-25152,746,-28667,-1938
C03206=3047,34992,-25073,755,-28691,-1910
C03207=2876,34919,-25163,780,-28662,-1844
C03208=2720,34820,-25285,802,-28623,-1783
C03209=2596,34672,-25466,821,-28566,-1736
C03210=2467,34521,-25649,840,-28509,-1686
C03211=2334,34377,-25825,860,-28453,-1635
C03212=2214,34218,-26018,879,-28393,-1589
C03213=2114,34054,-26217,894,-28331,-1551
C03214=1957,33990,-26297,917,-28305,-1490
C03215=1817,33867,-26447,938,-28258,-1436
C03216=1799,33682,-26671,943,-28189,-1430
C03217=1856,33512,-26875,937,-28127,-1454
C03218=1856,33512,-25475,937,-28127,-1454
C03219=2023,34057,-22215,907,-28331,-1515
C03220=2023,34057,-26215,907,-28331,-1515
C03221=2124,34118,-26140,892,-28355,-1554
C03222=2185,34235,-25998,883,-28399,-1577
C03223=2267,34347,-25862,870,-28441,-1609
C03224=2359,34450,-25736,856,-28481,-1644
C03225=2451,34553,-25610,842,-28520,-1679
C03226=2542,34657,-25484,829,-28560,-1714
C03227=2623,34767,-25350,816,-28602,-1746
C03228=2661,34849,-25250,810,-28633,-1760
C03229=2528,34839,-25264,829,-28627,-1708
C03230=2398,34839,-25265,847,-28626,-1657
C03231=2271,34849,-25255,864,-28628,-1607
C03232=2146,34863,-25239,882,-28631,-1558
C03233=2028,34901,-25194,898,-28644,-1511
C03234=1922,34976,-25105,911,-28670,-1469
C03235=1864,35083,-24976,918,-28709,-1445
C03236=1838,35210,-24824,921,-28755,-1434
C03237=1765,35218,-24814,931,-28757,-1405
C03238=1727,35096,-24962,937,-28711,-1391
C03239=1746,34966,-25119,936,-28664,-1400
C03240=1783,34846,-25264,932,-28620,-1415
C03241=1867,34753,-25375,921,-28587,-1449
C03242=1945,34657,-25490,912,-28552,-1480
C03243=1948,34618,-25537,912,-28538,-1482
C03244=1871,34715,-25421,921,-28572,-1451
C03245=1787,34807,-25310,932,-28605,-1417
C03246=1735,34919,-25176,938,-28646,-1396
C03247=1711,35046,-25023,940,-28693,-1386
C03248=1658,34997,-25083,948,-28674,-1365
C03249=1658,34864,-25243,949,-28625,-1366
C03250=1659,34732,-25403,951,-28576,-1367
C03251=1742,34638,-25515,940,-28542,-1401
C03252=1828,34547,-25625,929,-28510,-1435
C03253=1911,34453,-25737,919,-28476,-1469
C03254=1874,34455,-25735,924,-28476,-1454
C03255=1790,34548,-25624,934,-28510,-1420
C03256=1705,34640,-25513,945,-28542,-1386
C03257=1639,34743,-25390,953,-28580,-1359
C03258=1639,34868,-25239,952,-28626,-1358
C03259=1583,34847,-25265,960,-28617,-1337
C03260=1554,34722,-25416,965,-28571,-1326
C03261=1563,34595,-25570,965,-28524,-1331
C03262=1606,34478,-25710,961,-28481,-1349
C03263=1697,34390,-25816,949,-28450,-1385
C03264=1795,34305,-25918,936,-28420,-1424
C03265=1858,34229,-26009,928,-28392,-1449
C03266=1758,34307,-25916,942,-28420,-1409
C03267=1658,34385,-25822,955,-28447,-1370
C03268=1567,34474,-25716,966,-28479,-1333
C03269=1534,34596,-25569,969,-28524,-1320
C03270=1534,34728,-25409,968,-28573,-1318
C03271=1519,34805,-25316,969,-28601,-1312
C03272=1470,34685,-25462,977,-28556,-1294
C03273=1440,34560,-25613,983,-28509,-1283
C03274=1460,34430,-25770,982,-28461,-1292
C03275=1487,34305,-25921,979,-28416,-1303
C03276=1545,34197,-26050,972,-28376,-1327
C03277=1659,34147,-26110,957,-28359,-1372
C03278=1780,34117,-26145,940,-28350,-1420
C03279=1899,34077,-26192,924,-28337,-1466
C03280=2023,34057,-26215,907,-28331,-1515
C03281=2023,34057,-24815,907,-28331,-1515
C03282=1111,34448,-21752,1030,-28464,-1155
C03283=1111,34448,-25752,1030,-28464,-1155
C03284=1089,34435,-25767,1033,-28458,-1146
C03285=1065,34424,-25782,1036,-28454,-1137
C03286=1039,34419,-25788,1040,-28452,-1127
C03287=1016,34406,-25804,1043,-28447,-1118
C03288=992,34396,-25816,1047,-28443,-1108
C03289=967,34389,-25825,1051,-28440,-1098
C03290=944,34376,-25841,1054,-28435,-1090
C03291=917,34372,-25846,1058,-28433,-1079
C03292=895,34359,-25862,1061,-28428,-1070
C03293=867,34355,-25867,1065,-28426,-1060
C03294=840,34351,-25872,1069,-28424,-1049
C03295=813,34347,-25877,1072,-28422,-1039
C03296=786,34343,-25882,1076,-28420,-1028
C03297=759,34339,-25887,1080,-28418,-1017
C03298=732,34335,-25893,1084,-28417,-1007
C03299=708,34341,-25886,1087,-28418,-997
C03300=684,34346,-25880,1090,-28420,-988
C03301=657,34343,-25884,1094,-28419,-977
C03302=633,34349,-25877,1097,-28420,-968
C03303=608,34352,-25874,1101,-28421,-958
C03304=583,34354,-25872,1104,-28422,-948
C03305=560,34363,-25861,1107,-28425,-939
C03306=538,34372,-25850,1110,-28428,-930
C03307=515,34379,-25841,1113,-28430,-921
C03308=492,34390,-25829,1116,-28434,-912
C03309=470,34399,-25818,1119,-28437,-903
C03310=447,34408,-25807,1122,-28440,-894
C03311=427,34424,-25788,1125,-28445,-886
C03312=404,34433,-25777,1128,-28448,-877
C03313=396,34457,-25749,1129,-28457,-874
C03314=419,34449,-25759,1126,-28454,-883
C03315=440,34435,-25775,1123,-28450,-891
C03316=462,34424,-25789,1120,-28446,-900
C03317=484,34413,-25801,1117,-28442,-909
C03318=507,34405,-25810,1114,-28440,-918
C03319=528,34391,-25827,1111,-28434,-926
C03320=551,34385,-25834,1108,-28433,-936
C03321=575,34379,-25841,1105,-28431,-945
C03322=599,34373,-25848,1102,-28429,-954
C03323=623,34367,-24456,1099,-28427,-964
C03324=-41004,59868,4099,4900,-34257,16705
C03325=-41004,59868,1099,4900,-34257,16705
C03326=-41004,64596,1380,5213,-31659,16463
C03327=-41004,59868,1099,4900,-34257,16705
C03328=-41004,59868,9099,4900,-34257,16705
C03329=623,34367,-21856,1099,-28427,-964
C03330=623,34367,-25856,1099,-28427,-964
C03331=646,34361,-25863,1095,-28425,-973
C03332=673,34363,-25859,1092,-28426,-983
C03333=697,34359,-25864,1088,-28425,-993
C03334=724,34363,-25859,1085,-28427,-1004
C03335=748,34357,-25866,1081,-28425,-1013
C03336=775,34361,-25861,1077,-28427,-1024
C03337=803,34365,-25856,1074,-28428,-1034
C03338=830,34369,-25851,1070,-28430,-1045
C03339=857,34373,-25846,1066,-28432,-1055
C03340=884,34377,-25841,1062,-28434,-1066
C03341=908,34386,-25829,1059,-28438,-1076
C03342=934,34393,-25820,1055,-28441,-1085
C03343=957,34405,-25806,1052,-28445,-1095
C03344=983,34410,-25799,1048,-28448,-1105
C03345=1006,34423,-25783,1045,-28453,-1114
C03346=1030,34432,-25772,1041,-28457,-1123
C03347=1055,34440,-25762,1038,-28460,-1133
C03348=1078,34453,-25746,1034,-28465,-1142
C03349=1105,34457,-25741,1031,-28467,-1152
C03350=1111,34448,-25752,1030,-28464,-1155
C03351=1111,34448,-24352,1030,-28464,-1155
C03352=1082,34578,-21596,1032,-28511,-1142
C03353=1082,34578,-25596,1032,-28511,-1142
C03354=1056,34583,-25589,1036,-28513,-1132
C03355=1026,34579,-25595,1040,-28511,-1120
C03356=999,34585,-25588,1044,-28512,-1110
C03357=971,34585,-25588,1048,-28512,-1099
C03358=943,34586,-25587,1051,-28512,-1087
C03359=916,34592,-25581,1055,-28514,-1077
C03360=887,34589,-25584,1059,-28512,-1066
C03361=860,34593,-25580,1063,-28513,-1055
C03362=833,34598,-25573,1066,-28515,-1044
C03363=807,34604,-25567,1070,-28517,-1034
C03364=778,34604,-25568,1074,-28516,-1023
C03365=751,34607,-25564,1078,-28517,-1012
C03366=724,34611,-25560,1081,-28518,-1001
C03367=698,34617,-25553,1085,-28520,-991
C03368=671,34622,-25547,1089,-28522,-980
C03369=645,34628,-25540,1092,-28523,-970
C03370=618,34632,-25535,1096,-28525,-959
C03371=591,34636,-25531,1100,-28526,-949
C03372=564,34640,-25527,1103,-28527,-938
C03373=536,34643,-25523,1107,-28528,-927
C03374=509,34647,-25519,1111,-28529,-917
C03375=485,34658,-25506,1114,-28532,-907
C03376=458,34661,-25502,1118,-28533,-896
C03377=430,34665,-25498,1121,-28534,-885
C03378=406,34676,-25485,1125,-28538,-876
C03379=379,34679,-25481,1128,-28539,-865
C03380=354,34690,-25468,1132,-28542,-855
C03381=335,34698,-25459,1134,-28545,-848
C03382=353,34700,-25456,1132,-28546,-855
C03383=379,34694,-25464,1128,-28544,-865
C03384=405,34688,-25470,1125,-28542,-875
C03385=432,34682,-25477,1121,-28540,-886
C03386=459,34679,-25481,1117,-28539,-896
C03387=486,34675,-25485,1114,-28539,-907
C03388=513,34671,-25489,1110,-28538,-918
C03389=537,34661,-25502,1107,-28534,-928
C03390=565,34657,-25506,1103,-28533,-938
C03391=592,34653,-25510,1099,-28532,-949
C03392=619,34650,-25514,1096,-28531,-960
C03393=646,34646,-25518,1092,-28530,-970
C03394=673,34642,-25523,1088,-28529,-981
C03395=699,34636,-25530,1085,-28527,-991
C03396=726,34630,-25536,1081,-28525,-1002
C03397=752,34625,-25543,1077,-28524,-1012
C03398=782,34628,-25539,1073,-28525,-1024
C03399=809,34623,-25544,1070,-28524,-1034
C03400=835,34618,-25550,1066,-28522,-1045
C03401=862,34612,-25557,1062,-28521,-1055
C03402=888,34606,-25563,1059,-28519,-1066
C03403=918,34610,-25559,1055,-28520,-1077
C03404=944,34605,-25564,1051,-28519,-1088
C03405=972,34602,-25567,1047,-28519,-1099
C03406=1001,34604,-25565,1043,-28520,-1110
C03407=1027,34598,-25571,1040,-28518,-1121
C03408=1056,34599,-25571,1036,-28518,-1132
C03409=1084,34597,-25572,1032,-28518,-1143
C03410=1110,34592,-25579,1028,-28516,-1153
C03411=1138,34588,-25583,1024,-28515,-1164
C03412=1112,34582,-25590,1028,-28513,-1154
C03413=1082,34578,-25596,1032,-28511,-1142
C03414=1082,34578,-24196,1032,-28511,-1142
C03415=1146,34769,-21364,1021,-28582,-1166
C03416=1146,34769,-25364,1021,-28582,-1166
C03417=1111,34783,-25348,1026,-28587,-1152
C03418=1077,34797,-25331,1030,-28592,-1138
C03419=1042,34811,-25315,1035,-28596,-1125
C03420=1008,34825,-25298,1040,-28601,-1111
C03421=974,34842,-25277,1044,-28607,-1098
C03422=941,34860,-25256,1048,-28613,-1084
C03423=908,34878,-25235,1053,-28619,-1071
C03424=874,34895,-25215,1057,-28625,-1058
C03425=841,34913,-25194,1062,-28631,-1045
C03426=810,34937,-25164,1065,-28640,-1032
C03427=777,34955,-25144,1070,-28646,-1019
C03428=743,34973,-25123,1074,-28652,-1006
C03429=713,34997,-25093,1078,-28661,-993
C03430=679,35015,-25072,1083,-28667,-980
C03431=649,35040,-25043,1086,-28675,-968
C03432=615,35057,-25022,1091,-28681,-955
C03433=585,35082,-24993,1095,-28690,-942
C03434=554,35107,-24963,1099,-28699,-930
C03435=523,35131,-24934,1103,-28707,-918
C03436=493,35156,-24904,1106,-28716,-906
C03437=468,35185,-24870,1109,-28726,-896
C03438=438,35209,-24841,1113,-28735,-884
C03439=407,35234,-24811,1117,-28743,-871
C03440=383,35262,-24777,1120,-28754,-862
C03441=359,35291,-24743,1123,-28764,-852
C03442=337,35321,-24708,1126,-28774,-843
C03443=316,35351,-24671,1128,-28785,-834
C03444=295,35381,-24635,1131,-28796,-826
C03445=276,35412,-24597,1133,-28807,-818
C03446=281,35436,-24569,1132,-28816,-820
C03447=298,35403,-24608,1130,-28804,-827
C03448=322,35375,-24642,1127,-28794,-837
C03449=340,35343,-24681,1125,-28782,-844
C03450=364,35314,-24715,1122,-28772,-853
C03451=388,35286,-24749,1119,-28762,-863
C03452=412,35257,-24783,1116,-28752,-873
C03453=443,35232,-24813,1112,-28743,-885
C03454=467,35204,-24846,1109,-28733,-895
C03455=497,35179,-24876,1105,-28725,-907
C03456=528,35155,-24906,1102,-28716,-920
C03457=559,35130,-24935,1098,-28707,-932
C03458=589,35105,-24965,1094,-28699,-944
C03459=620,35080,-24994,1090,-28690,-956
C03460=653,35063,-25015,1085,-28684,-970
C03461=684,35038,-25044,1082,-28675,-982
C03462=717,35021,-25065,1077,-28669,-995
C03463=748,34996,-25095,1073,-28661,-1007
C03464=781,34978,-25115,1069,-28655,-1021
C03465=814,34959,-25139,1065,-28648,-1034
C03466=846,34936,-25166,1061,-28640,-1046
C03467=879,34918,-25187,1056,-28634,-1060
C03468=912,34901,-25207,1052,-28628,-1073
C03469=945,34883,-25228,1047,-28622,-1086
C03470=979,34866,-25249,1043,-28616,-1099
C03471=1012,34848,-25270,1039,-28610,-1113
C03472=1046,34830,-25291,1034,-28604,-1126
C03473=1079,34813,-25312,1030,-28598,-1139
C03474=1115,34802,-25324,1025,-28594,-1153
C03475=1148,34785,-25345,1021,-28588,-1166
C03476=1146,34769,-25364,1021,-28582,-1166
C03477=1146,34769,-23964,1021,-28582,-1166
C03478=1388,34961,-21129,985,-28657,-1259
C03479=1388,34961,-25129,985,-28657,-1259
C03480=1355,34978,-25109,990,-28663,-1246
C03481=1321,34996,-25088,994,-28669,-1233
C03482=1290,35021,-25058,998,-28677,-1220
C03483=1257,35038,-25037,1003,-28683,-1207
C03484=1225,35063,-25008,1007,-28692,-1195
C03485=1194,35088,-24979,1011,-28701,-1182
C03486=1161,35105,-24958,1015,-28707,-1169
C03487=1130,35130,-24928,1019,-28716,-1157
C03488=1097,35147,-24907,1023,-28722,-1143
C03489=1066,35172,-24878,1027,-28730,-1131
C03490=1035,35197,-24848,1031,-28739,-1119
C03491=1004,35222,-24819,1035,-28748,-1106
C03492=973,35246,-24790,1039,-28756,-1094
C03493=940,35264,-24769,1044,-28762,-1081
C03494=909,35289,-24739,1048,-28771,-1068
C03495=878,35313,-24710,1051,-28780,-1056
C03496=847,35338,-24680,1055,-28788,-1044
C03497=814,35356,-24659,1060,-28794,-1030
C03498=784,35380,-24630,1064,-28803,-1018
C03499=753,35405,-23201,1068,-28812,-1006
C03500=-41004,59868,4099,4900,-34257,16705
C03501=-41004,59868,1099,4900,-34257,16705
C03502=-41004,64596,1380,5213,-31659,16463
C03503=-41004,59868,1099,4900,-34257,16705
C03504=-41004,59868,9099,4900,-34257,16705
C03505=753,35405,-20601,1068,-28812,-1006
C03506=753,35405,-24601,1068,-28812,-1006
C03507=722,35430,-24571,1071,-28820,-994
C03508=691,35454,-24542,1075,-28829,-981
C03509=661,35479,-24512,1079,-28838,-969
C03510=628,35497,-24491,1084,-28844,-956
C03511=597,35522,-24462,1087,-28852,-944
C03512=564,35539,-24441,1092,-28858,-930
C03513=531,35557,-24420,1096,-28864,-917
C03514=499,35574,-24399,1100,-28870,-904
C03515=501,35591,-24380,1100,-28876,-905
C03516=535,35576,-24396,1095,-28872,-919
C03517=569,35562,-24413,1091,-28867,-932
C03518=600,35538,-24442,1087,-28858,-944
C03519=633,35520,-24463,1083,-28852,-957
C03520=665,35502,-24484,1078,-28846,-971
C03521=696,35478,-24514,1074,-28838,-983
C03522=727,35453,-24543,1071,-28829,-995
C03523=757,35428,-24572,1067,-28820,-1007
C03524=790,35411,-24593,1062,-28814,-1021
C03525=821,35386,-24623,1058,-28806,-1033
C03526=852,35361,-24652,1054,-28797,-1045
C03527=883,35336,-24682,1051,-28788,-1058
C03528=914,35312,-24711,1047,-28780,-1070
C03529=946,35293,-24733,1042,-28773,-1083
C03530=978,35269,-24761,1038,-28765,-1095
C03531=1008,35245,-24791,1034,-28756,-1108
C03532=1039,35220,-24820,1030,-28747,-1120
C03533=1070,35195,-24850,1026,-28739,-1133
C03534=1102,35173,-24876,1022,-28731,-1145
C03535=1135,35153,-24900,1018,-28724,-1158
C03536=1166,35128,-24930,1014,-28715,-1171
C03537=1197,35104,-24959,1010,-28707,-1183
C03538=1230,35086,-24980,1006,-28701,-1196
C03539=1261,35061,-25009,1002,-28692,-1209
C03540=1294,35044,-25030,997,-28686,-1222
C03541=1326,35019,-25060,993,-28677,-1234
C03542=1359,35001,-25081,989,-28671,-1248
C03543=1390,34977,-25110,985,-28663,-1260
C03544=1424,34959,-25131,981,-28657,-1273
C03545=1422,34943,-25150,981,-28651,-1273
C03546=1388,34961,-25129,985,-28657,-1259
C03547=1388,34961,-23729,985,-28657,-1259
C03548=1511,35406,-20590,963,-28823,-1304
C03549=1511,35406,-24590,963,-28823,-1304
C03550=1486,35425,-24567,967,-28830,-1294
C03551=1462,35445,-24543,970,-28837,-1285
C03552=1437,35465,-24520,973,-28844,-1275
C03553=1412,35484,-24497,976,-28851,-1265
C03554=1394,35508,-24469,978,-28859,-1257
C03555=1369,35527,-24445,982,-28866,-1248
C03556=1351,35551,-24417,984,-28874,-1240
C03557=1333,35574,-24389,986,-28883,-1233
C03558=1308,35594,-24366,989,-28890,-1223
C03559=1290,35617,-24337,991,-28898,-1216
C03560=1266,35637,-24314,994,-28905,-1206
C03561=1248,35660,-24286,997,-28913,-1199
C03562=1225,35681,-24261,1000,-28920,-1189
C03563=1205,35703,-24234,1002,-28929,-1181
C03564=1183,35725,-24209,1005,-28936,-1173
C03565=1163,35747,-24183,1007,-28944,-1165
C03566=1144,35770,-24155,1010,-28952,-1157
C03567=1126,35793,-24127,1012,-28961,-1150
C03568=1108,35817,-24099,1014,-28969,-1142
C03569=1090,35840,-24071,1016,-28977,-1135
C03570=1066,35860,-24047,1019,-28984,-1125
C03571=1048,35883,-24019,1021,-28993,-1118
C03572=1030,35907,-23991,1024,-29001,-1111
C03573=1012,35930,-23963,1026,-29009,-1104
C03574=994,35954,-23935,1028,-29018,-1096
C03575=976,35977,-23907,1030,-29026,-1089
C03576=956,35999,-23880,1032,-29034,-1081
C03577=934,36020,-23855,1035,-29041,-1072
C03578=916,36043,-23827,1038,-29050,-1065
C03579=924,36055,-23814,1036,-29054,-1068
C03580=945,36033,-23840,1034,-29046,-1076
C03581=967,36011,-23865,1031,-29039,-1085
C03582=985,35989,-23893,1029,-29031,-1093
C03583=1006,35967,-23919,1026,-29023,-1101
C03584=1026,35945,-23945,1024,-29015,-1109
C03585=1045,35922,-23973,1021,-29007,-1117
C03586=1063,35898,-24001,1019,-28998,-1124
C03587=1081,35875,-24029,1017,-28990,-1131
C03588=1099,35851,-24057,1015,-28982,-1138
C03589=1119,35829,-24084,1012,-28974,-1147
C03590=1140,35807,-24110,1010,-28966,-1155
C03591=1159,35785,-24137,1007,-28958,-1163
C03592=1177,35761,-24165,1005,-28949,-1170
C03593=1195,35738,-24193,1003,-28941,-1177
C03594=1220,35718,-24216,1000,-28934,-1187
C03595=1238,35695,-24244,998,-28926,-1195
C03596=1256,35671,-24273,995,-28917,-1202
C03597=1281,35652,-24296,992,-28911,-1212
C03598=1299,35628,-24324,990,-28902,-1219
C03599=1323,35609,-24347,987,-28895,-1229
C03600=1342,35585,-24376,985,-28887,-1236
C03601=1366,35565,-24399,982,-28880,-1246
C03602=1384,35542,-24427,979,-28872,-1253
C03603=1407,35521,-24452,976,-28864,-1262
C03604=1427,35499,-24478,974,-28856,-1271
C03605=1452,35480,-24502,971,-28849,-1280
C03606=1470,35456,-24530,969,-28841,-1288
C03607=1495,35436,-24553,965,-28834,-1298
C03608=1520,35417,-24577,962,-28827,-1308
C03609=1511,35406,-24590,963,-28823,-1304
C03610=1511,35406,-23190,963,-28823,-1304
C03611=1780,35509,-20463,925,-28865,-1409
C03612=1780,35509,-24463,925,-28865,-1409
C03613=1762,35535,-24431,928,-28874,-1402
C03614=1742,35559,-24402,930,-28883,-1394
C03615=1726,35586,-24370,932,-28893,-1387
C03616=1709,35612,-24338,934,-28902,-1381
C03617=1689,35637,-24309,936,-28911,-1373
C03618=1669,35662,-24279,939,-28920,-1365
C03619=1651,35687,-24248,941,-28929,-1357
C03620=1636,35715,-24216,943,-28939,-1351
C03621=1616,35739,-24186,945,-28948,-1343
C03622=1598,35765,-24156,948,-28957,-1336
C03623=1577,35789,-24127,950,-28966,-1327
C03624=1563,35817,-24093,952,-28976,-1322
C03625=1544,35842,-24063,954,-28985,-1314
C03626=1533,35871,-24027,955,-28996,-1309
C03627=1517,35898,-23995,957,-29005,-1303
C03628=1500,35925,-23963,959,-29015,-1296
C03629=1488,35954,-23928,960,-29025,-1291
C03630=1477,35983,-23893,962,-29036,-1286
C03631=1457,36008,-23863,964,-29045,-1278
C03632=1444,36037,-23829,966,-29055,-1273
C03633=1433,36066,-23793,967,-29066,-1268
C03634=1421,36095,-23758,968,-29077,-1263
C03635=1409,36125,-23723,969,-29087,-1259
C03636=1398,36154,-23688,971,-29098,-1254
C03637=1401,36178,-23659,970,-29107,-1255
C03638=1417,36151,-23691,968,-29097,-1261
C03639=1428,36122,-23726,967,-29087,-1266
C03640=1440,36093,-23761,966,-29076,-1271
C03641=1454,36064,-23795,964,-29066,-1277
C03642=1467,36036,-23829,963,-29055,-1282
C03643=1484,36010,-23861,960,-29046,-1289
C03644=1496,35981,-23896,959,-29035,-1294
C03645=1507,35951,-23931,958,-29025,-1299
C03646=1526,35926,-23961,956,-29016,-1306
C03647=1540,35898,-23995,954,-29005,-1312
C03648=1553,35869,-24030,953,-28995,-1317
C03649=1566,35841,-24064,951,-28985,-1323
C03650=1584,35815,-24095,949,-28976,-1330
C03651=1605,35791,-24123,946,-28967,-1338
C03652=1619,35763,-24157,945,-28957,-1344
C03653=1639,35739,-24186,942,-28948,-1352
C03654=1659,35714,-24216,940,-28939,-1360
C03655=1672,35686,-24250,938,-28929,-1366
C03656=1692,35661,-24280,936,-28920,-1374
C03657=1712,35636,-24309,933,-28911,-1382
C03658=1732,35612,-24339,931,-28902,-1390
C03659=1746,35583,-24373,929,-28892,-1395
C03660=1766,35559,-24402,927,-28883,-1403
C03661=1785,35534,-24432,924,-28875,-1411
C03662=1805,35510,-24461,922,-28866,-1419
C03663=1820,35482,-24495,920,-28856,-1425
C03664=1839,35457,-24525,918,-28847,-1433
C03665=1859,35432,-24554,915,-28838,-1441
C03666=1874,35405,-24587,914,-28828,-1447
C03667=1876,35383,-24613,914,-28820,-1448
C03668=1856,35408,-24584,916,-28829,-1440
C03669=1836,35433,-24554,919,-28838,-1432
C03670=1822,35461,-24520,920,-28848,-1426
C03671=1801,35485,-24492,923,-28856,-1418
C03672=1780,35509,-23063,925,-28865,-1409
C03673=-41004,59868,4099,4900,-34257,16705
C03674=-41004,59868,1099,4900,-34257,16705
C03675=-41004,64596,1380,5213,-31659,16463
C03676=-41004,59868,1099,4900,-34257,16705
C03677=-41004,59868,9099,4900,-34257,16705
C03678=1780,35509,-20463,925,-28865,-1409
C03679=1780,35509,-24463,925,-28865,-1409
C03680=1780,35509,-23063,925,-28865,-1409
C03681=2074,35525,-20439,885,-28875,-1525
C03682=2074,35525,-24439,885,-28875,-1525
C03683=2071,35554,-24404,885,-28886,-1524
C03684=2060,35578,-24376,886,-28895,-1519
C03685=2057,35607,-24341,886,-28905,-1518
C03686=2055,35636,-24306,886,-28916,-1517
C03687=2053,35665,-24271,886,-28927,-1515
C03688=2050,35694,-24236,886,-28938,-1514
C03689=2048,35723,-24201,886,-28948,-1513
C03690=2045,35752,-24166,886,-28959,-1512
C03691=2043,35781,-24131,886,-28970,-1511
C03692=2031,35804,-24102,888,-28978,-1506
C03693=2029,35833,-24067,888,-28989,-1505
C03694=2026,35862,-24032,888,-29000,-1504
C03695=2024,35891,-23997,888,-29010,-1503
C03696=2021,35920,-23962,888,-29021,-1501
C03697=2010,35944,-23934,889,-29030,-1497
C03698=2007,35973,-23899,889,-29040,-1495
C03699=2005,36002,-23864,889,-29051,-1494
C03700=1993,36026,-23835,891,-29060,-1490
C03701=1991,36054,-23800,891,-29070,-1488
C03702=1986,36082,-23767,891,-29080,-1486
C03703=1977,36107,-23737,892,-29090,-1483
C03704=1975,36136,-23702,892,-29100,-1481
C03705=1972,36165,-23667,892,-29111,-1480
C03706=1961,36189,-23638,894,-29120,-1476
C03707=1958,36218,-23603,894,-29130,-1474
C03708=1947,36241,-23575,895,-29139,-1470
C03709=1950,36260,-23553,894,-29146,-1471
C03710=1959,36235,-23583,893,-29137,-1475
C03711=1968,36210,-23613,892,-29127,-1479
C03712=1980,36186,-23641,891,-29119,-1483
C03713=1982,36157,-23676,891,-29108,-1484
C03714=1990,36131,-23708,890,-29099,-1488
C03715=1996,36104,-23740,890,-29089,-1490
C03716=1999,36075,-23775,890,-29078,-1491
C03717=2010,36052,-23803,888,-29070,-1496
C03718=2013,36023,-23838,888,-29059,-1497
C03719=2023,35999,-23867,887,-29050,-1502
C03720=2027,35970,-23902,887,-29040,-1503
C03721=2029,35941,-23937,887,-29029,-1504
C03722=2039,35916,-23967,886,-29020,-1508
C03723=2043,35889,-24000,885,-29010,-1510
C03724=2045,35860,-24035,885,-28999,-1511
C03725=2048,35831,-24070,885,-28988,-1512
C03726=2050,35802,-24105,885,-28977,-1514
C03727=2059,35776,-24135,884,-28968,-1517
C03728=2064,35749,-24169,884,-28958,-1519
C03729=2067,35720,-24204,884,-28947,-1521
C03730=2069,35691,-24239,884,-28937,-1522
C03731=2072,35662,-24274,884,-28926,-1523
C03732=2074,35633,-24309,884,-28915,-1524
C03733=2077,35604,-24344,884,-28905,-1525
C03734=2079,35575,-24379,884,-28894,-1527
C03735=2082,35546,-24414,884,-28883,-1528
C03736=2093,35523,-24442,882,-28875,-1532
C03737=2096,35494,-24477,882,-28864,-1534
C03738=2098,35465,-24512,882,-28853,-1535
C03739=2090,35444,-24537,883,-28845,-1532
C03740=2081,35469,-24507,884,-28855,-1528
C03741=2076,35496,-24474,885,-28865,-1526
C03742=2074,35525,-24439,885,-28875,-1525
C03743=2074,35525,-23039,885,-28875,-1525
C03744=2577,35564,-20387,815,-28897,-1722
C03745=2577,35564,-24387,815,-28897,-1722
C03746=2574,35595,-24349,815,-28908,-1721
C03747=2581,35624,-24314,814,-28919,-1723
C03748=2588,35652,-24279,813,-28930,-1726
C03749=2594,35681,-24245,812,-28941,-1728
C03750=2601,35710,-24209,811,-28952,-1731
C03751=2607,35739,-24174,809,-28962,-1733
C03752=2613,35768,-24139,808,-28973,-1735
C03753=2619,35797,-24104,807,-28984,-1737
C03754=2619,35827,-24068,807,-28995,-1737
C03755=2631,35854,-24034,805,-29006,-1742
C03756=2637,35883,-23999,804,-29016,-1744
C03757=2643,35912,-23964,803,-29027,-1746
C03758=2656,35939,-23931,801,-29038,-1751
C03759=2662,35968,-23896,800,-29048,-1753
C03760=2669,35997,-23862,799,-29059,-1756
C03761=2681,36024,-23828,797,-29069,-1761
C03762=2693,36052,-23795,795,-29080,-1765
C03763=2707,36078,-23762,793,-29090,-1770
C03764=2716,36106,-23728,791,-29100,-1774
C03765=2732,36133,-23696,789,-29110,-1780
C03766=2746,36160,-23663,787,-29121,-1785
C03767=2759,36187,-23630,785,-29131,-1790
C03768=2778,36212,-23600,782,-29141,-1798
C03769=2798,36237,-23569,779,-29150,-1805
C03770=2818,36263,-23538,776,-29160,-1813
C03771=2837,36288,-23507,773,-29170,-1820
C03772=2860,36307,-23484,770,-29177,-1829
C03773=2883,36327,-23460,766,-29185,-1838
C03774=2906,36345,-23437,763,-29192,-1847
C03775=2934,36348,-23432,759,-29194,-1858
C03776=2919,36332,-23453,761,-29187,-1853
C03777=2894,36318,-23470,765,-29182,-1842
C03778=2872,36296,-23496,768,-29173,-1834
C03779=2851,36274,-23524,771,-29165,-1826
C03780=2830,36252,-23551,774,-29156,-1818
C03781=2815,36227,-23580,777,-29147,-1812
C03782=2795,36202,-23611,779,-29137,-1804
C03783=2776,36177,-23642,782,-29128,-1797
C03784=2763,36150,-23675,784,-29117,-1792
C03785=2743,36124,-23706,787,-29108,-1784
C03786=2730,36097,-23739,789,-29097,-1779
C03787=2719,36070,-23773,791,-29087,-1775
C03788=2711,36041,-23807,792,-29076,-1772
C03789=2698,36014,-23840,794,-29066,-1767
C03790=2689,35986,-23874,796,-29055,-1764
C03791=2679,35958,-23908,797,-29045,-1760
C03792=2666,35931,-23941,800,-29035,-1755
C03793=2660,35902,-23976,801,-29024,-1753
C03794=2653,35874,-24010,802,-29013,-1750
C03795=2646,35845,-24045,803,-29002,-1748
C03796=2639,35816,-24080,804,-28992,-1745
C03797=2632,35788,-24115,806,-28981,-1743
C03798=2625,35759,-24150,807,-28970,-1740
C03799=2618,35730,-24184,808,-28959,-1738
C03800=2612,35702,-24219,809,-28949,-1735
C03801=2605,35673,-24254,810,-28938,-1733
C03802=2599,35644,-24289,811,-28927,-1730
C03803=2592,35615,-24324,813,-28916,-1728
C03804=2593,35584,-24361,813,-28905,-1729
C03805=2577,35564,-24387,815,-28897,-1722
C03806=2577,35564,-22987,815,-28897,-1722
C03807=2999,35837,-20051,755,-29004,-1887
C03808=2999,35837,-24051,755,-29004,-1887
C03809=3018,35859,-24025,752,-29013,-1894
C03810=3045,35874,-24005,748,-29019,-1905
C03811=3070,35895,-23980,744,-29027,-1914
C03812=3099,35909,-23963,740,-29033,-1925
C03813=3127,35923,-23946,736,-29038,-1937
C03814=3158,35933,-23932,732,-29043,-1949
C03815=3189,35942,-23921,728,-29046,-1961
C03816=3217,35957,-23903,724,-29052,-1972
C03817=3247,35969,-23888,720,-29057,-1983
C03818=3275,35983,-23871,715,-29063,-1995
C03819=3304,35997,-23854,711,-29068,-2006
C03820=3333,36010,-23837,707,-29074,-2017
C03821=3361,36024,-23820,703,-29079,-2028
C03822=3390,36038,-23803,699,-29085,-2039
C03823=3418,36052,-23785,695,-29091,-2050
C03824=3447,36066,-23768,691,-29096,-2062
C03825=3473,36083,-23747,688,-29103,-2072
C03826=3501,36098,-23728,684,-29109,-2083
C03827=3528,36116,-23707,680,-29116,-2093
C03828=3556,36130,-23689,676,-29122,-2104
C03829=3582,36149,-23666,672,-29129,-2114
C03830=3610,36163,-23648,668,-29135,-2125
C03831=3637,36180,-23628,664,-29142,-2136
C03832=3662,36199,-23604,661,-29149,-2146
C03833=3687,36220,-23578,657,-29157,-2155
C03834=3712,36239,-23555,654,-29165,-2165
C03835=3739,36256,-23534,650,-29171,-2176
C03836=3763,36277,-23509,646,-29180,-2185
C03837=3788,36298,-23483,643,-29188,-2195
C03838=3810,36316,-23461,640,-29195,-2203
C03839=3798,36290,-23492,641,-29185,-2199
C03840=3774,36269,-23518,645,-29177,-2189
C03841=3749,36248,-23544,648,-29169,-2180
C03842=3725,36227,-23570,652,-29160,-2170
C03843=3699,36208,-23592,656,-29153,-2160
C03844=3676,36186,-23620,659,-29144,-2151
C03845=3648,36170,-23639,663,-29138,-2140
C03846=3623,36149,-23665,666,-29130,-2131
C03847=3595,36136,-23682,670,-29124,-2120
C03848=3568,36120,-22302,674,-29118,-2109
C03849=-41004,59868,4099,4900,-34257,16705
C03850=-41004,59868,1099,4900,-34257,16705
C03851=-41004,64596,1380,5213,-31659,16463
C03852=-41004,59868,1099,4900,-34257,16705
C03853=-41004,59868,9099,4900,-34257,16705
C03854=3568,36120,-19702,674,-29118,-2109
C03855=3568,36120,-23702,674,-29118,-2109
C03856=3543,36099,-23727,678,-29110,-2099
C03857=3514,36085,-23744,682,-29104,-2088
C03858=3486,36071,-23761,686,-29099,-2077
C03859=3459,36054,-23782,690,-29092,-2066
C03860=3431,36040,-23800,694,-29086,-2056
C03861=3405,36021,-23823,697,-29079,-2045
C03862=3375,36010,-23837,702,-29074,-2034
C03863=3347,35995,-23855,706,-29068,-2023
C03864=3319,35980,-23873,710,-29063,-2012
C03865=3287,35972,-23884,714,-29059,-1999
C03866=3259,35957,-23902,718,-29053,-1988
C03867=3228,35947,-23915,722,-29049,-1976
C03868=3200,35933,-23932,726,-29043,-1965
C03869=3171,35920,-23949,730,-29038,-1954
C03870=3143,35906,-23966,734,-29032,-1943
C03871=3112,35896,-23978,739,-29028,-1931
C03872=3084,35881,-23996,743,-29022,-1920
C03873=3057,35864,-24017,747,-29016,-1909
C03874=3028,35850,-24034,751,-29010,-1898
C03875=2999,35837,-24051,755,-29004,-1887
C03876=2999,35837,-22651,755,-29004,-1887
C03877=3895,35774,-20117,632,-28994,-2239
C03878=3895,35774,-24117,632,-28994,-2239
C03879=3909,35807,-24077,630,-29006,-2244
C03880=3916,35841,-24035,628,-29019,-2247
C03881=3927,35874,-23994,627,-29032,-2252
C03882=3944,35907,-23955,624,-29044,-2258
C03883=3953,35940,-23914,623,-29057,-2261
C03884=3970,35973,-23875,620,-29069,-2268
C03885=3986,36005,-23836,618,-29081,-2274
C03886=4002,36037,-23797,615,-29093,-2280
C03887=4019,36069,-23758,613,-29106,-2287
C03888=4042,36099,-23721,609,-29117,-2296
C03889=4064,36130,-23683,606,-29129,-2304
C03890=4082,36162,-23645,603,-29141,-2311
C03891=4098,36194,-23605,601,-29153,-2317
C03892=4120,36224,-23568,598,-29165,-2326
C03893=4137,36256,-23529,595,-29177,-2332
C03894=4153,36288,-23490,593,-29189,-2339
C03895=4170,36320,-23451,590,-29202,-2345
C03896=4181,36354,-23411,588,-29214,-2349
C03897=4202,36384,-23373,585,-29226,-2357
C03898=4218,36417,-23334,583,-29238,-2363
C03899=4234,36449,-23295,581,-29251,-2370
C03900=4257,36479,-23258,577,-29262,-2379
C03901=4273,36511,-23219,575,-29274,-2385
C03902=4296,36541,-23182,572,-29286,-2394
C03903=4323,36565,-23152,568,-29295,-2404
C03904=4348,36592,-23119,564,-29306,-2414
C03905=4375,36615,-23091,560,-29315,-2424
C03906=4402,36637,-23064,556,-29324,-2435
C03907=4433,36650,-23048,552,-29329,-2447
C03908=4419,36628,-23075,554,-29320,-2442
C03909=4390,36608,-23100,558,-29312,-2431
C03910=4364,36585,-23128,562,-29303,-2420
C03911=4337,36562,-23156,566,-29294,-2410
C03912=4314,36531,-23193,569,-29283,-2401
C03913=4291,36501,-23230,573,-29271,-2392
C03914=4268,36471,-23267,576,-29259,-2383
C03915=4251,36439,-23306,578,-29247,-2377
C03916=4232,36408,-23344,581,-29235,-2369
C03917=4212,36376,-23382,584,-29223,-2361
C03918=4196,36344,-23422,586,-29211,-2355
C03919=4180,36312,-23461,589,-29199,-2349
C03920=4164,36280,-23500,591,-29187,-2343
C03921=4148,36248,-23539,594,-29174,-2336
C03922=4131,36216,-23578,596,-29162,-2330
C03923=4115,36184,-23617,599,-29150,-2324
C03924=4092,36154,-23654,602,-29138,-2315
C03925=4076,36121,-23693,604,-29126,-2309
C03926=4059,36089,-23732,607,-29114,-2303
C03927=4036,36059,-23769,610,-29102,-2293
C03928=4019,36027,-23808,613,-29090,-2287
C03929=3997,35997,-23846,616,-29078,-2278
C03930=3987,35963,-23887,618,-29066,-2275
C03931=3971,35931,-23926,620,-29053,-2268
C03932=3954,35899,-23965,623,-29041,-2262
C03933=3942,35865,-24005,625,-29029,-2257
C03934=3929,35833,-24045,627,-29016,-2252
C03935=3919,35799,-24086,628,-29003,-2249
C03936=3906,35766,-24126,630,-28991,-2244
C03937=3890,35739,-24159,633,-28981,-2237
C03938=3895,35774,-24117,632,-28994,-2239
C03939=3895,35774,-22717,632,-28994,-2239
C03940=4184,35297,-20691,595,-28820,-2355
C03941=4184,35297,-24691,595,-28820,-2355
C03942=3985,35217,-24790,623,-28787,-2278
C03943=3999,35079,-24957,622,-28736,-2284
C03944=4107,34904,-25169,609,-28672,-2327
C03945=4158,34700,-25415,603,-28597,-2347
C03946=4132,34721,-25390,606,-28605,-2337
C03947=4076,34927,-25141,613,-28681,-2314
C03948=3956,35095,-24939,628,-28742,-2266
C03949=3773,35147,-24877,653,-28759,-2194
C03950=3727,35027,-25024,661,-28713,-2177
C03951=3643,34831,-25261,674,-28639,-2145
C03952=3520,34644,-25489,692,-28568,-2098
C03953=3372,34469,-25703,714,-28501,-2041
C03954=3217,34305,-25902,738,-28438,-1981
C03955=3347,34362,-25833,719,-28461,-2032
C03956=3506,34519,-25641,695,-28521,-2093
C03957=3664,34676,-25450,672,-28582,-2154
C03958=3845,34674,-25450,647,-28583,-2225
C03959=3780,34480,-25686,657,-28510,-2201
C03960=3640,34303,-25902,678,-28442,-2147
C03961=3629,34175,-26056,681,-28395,-2143
C03962=3823,34252,-25961,653,-28426,-2219
C03963=3990,34391,-25792,629,-28480,-2283
C03964=4097,34494,-25666,613,-28519,-2325
C03965=3946,34324,-25872,635,-28454,-2267
C03966=3865,34223,-25996,647,-28416,-2235
C03967=4040,34324,-25871,622,-28456,-2303
C03968=4188,34494,-25664,600,-28521,-2360
C03969=4292,34685,-25431,584,-28593,-2400
C03970=4351,34884,-25191,575,-28668,-2422
C03971=4284,35083,-24950,583,-28742,-2395
C03972=4275,35146,-24873,583,-28765,-2392
C03973=4349,34950,-25110,574,-28693,-2421
C03974=4343,34750,-25353,577,-28618,-2420
C03975=4249,34556,-25588,591,-28545,-2384
C03976=4127,34380,-25803,610,-28477,-2337
C03977=3961,34237,-25978,634,-28422,-2273
C03978=4040,34210,-26010,623,-28413,-2304
C03979=4243,34290,-25911,594,-28445,-2383
C03980=4427,34401,-25775,567,-28489,-2454
C03981=4594,34541,-25603,543,-28543,-2519
C03982=4750,34698,-25412,520,-28604,-2579
C03983=4615,34525,-25623,540,-28538,-2527
C03984=4447,34387,-25791,564,-28484,-2462
C03985=4261,34281,-25922,591,-28442,-2390
C03986=4413,34208,-26009,570,-28417,-2450
C03987=4634,34211,-26003,539,-28421,-2536
C03988=4859,34237,-25970,507,-28433,-2624
C03989=5069,34304,-25886,477,-28460,-2706
C03990=5256,34408,-25758,450,-28502,-2779
C03991=5409,34570,-25561,428,-28564,-2838
C03992=5513,34760,-25329,413,-28636,-2878
C03993=5556,34965,-25080,406,-28714,-2894
C03994=5545,35183,-24816,406,-28795,-2889
C03995=5431,35356,-24606,421,-28859,-2844
C03996=5256,35472,-24468,445,-28900,-2775
C03997=5041,35478,-24462,475,-28899,-2691
C03998=4821,35465,-24481,505,-28891,-2604
C03999=4601,35423,-24534,536,-28873,-2518
C04000=4396,35354,-24620,565,-28844,-2438
C04001=4184,35297,-24691,595,-28820,-2355
C04002=4184,35297,-23291,595,-28820,-2355
C04003=4638,35127,-20892,533,-28763,-2534
C04004=4638,35127,-24892,533,-28763,-2534
C04005=4646,35125,-24895,532,-28762,-2537
C04006=4650,35111,-24911,531,-28757,-2538
C04007=4657,35100,-24925,530,-28753,-2541
C04008=4662,35087,-24941,530,-28748,-2544
C04009=4668,35075,-24956,529,-28743,-2546
C04010=4675,35063,-24970,528,-28739,-2549
C04011=4677,35048,-24987,528,-28734,-2549
C04012=4679,35034,-25005,528,-28728,-2550
C04013=4690,35024,-25017,526,-28725,-2554
C04014=4692,35010,-25034,526,-28719,-2555
C04015=4693,34995,-25052,526,-28714,-2556
C04016=4695,34980,-25070,526,-28708,-2557
C04017=4697,34965,-25088,526,-28703,-2558
C04018=4693,34952,-25104,526,-28698,-2556
C04019=4691,34939,-25121,527,-28693,-2555
C04020=4689,34925,-25137,527,-28688,-2555
C04021=4684,34912,-25153,528,-28683,-2553
C04022=4677,34899,-25169,529,-28678,-2550
C04023=4675,34885,-25185,529,-28673,-2549
C04024=4670,34872,-23801,530,-28668,-2547
C04025=-41004,59868,4099,4900,-34257,16705
C04026=-41004,59868,1099,4900,-34257,16705
C04027=-41004,64596,1380,5213,-31659,16463
C04028=-41004,59868,1099,4900,-34257,16705
C04029=-41004,59868,9099,4900,-34257,16705
C04030=4670,34872,-21201,530,-28668,-2547
C04031=4670,34872,-25201,530,-28668,-2547
C04032=4664,34860,-25217,531,-28663,-2545
C04033=4662,34846,-25233,531,-28658,-2544
C04034=4652,34834,-25248,533,-28653,-2541
C04035=4643,34822,-25262,534,-28649,-2537
C04036=4638,34809,-25278,535,-28644,-2535
C04037=4631,34796,-25294,536,-28639,-2533
C04038=4622,34784,-25308,537,-28634,-2529
C04039=4614,34772,-25323,539,-28630,-2526
C04040=4611,34759,-25339,539,-28625,-2525
C04041=4601,34747,-25354,540,-28620,-2521
C04042=4588,34741,-25361,542,-28618,-2516
C04043=4590,34755,-25344,542,-28623,-2517
C04044=4595,34768,-25328,541,-28628,-2518
C04045=4602,34780,-25313,540,-28633,-2521
C04046=4611,34792,-25299,539,-28637,-2525
C04047=4619,34805,-25284,538,-28642,-2528
C04048=4623,34818,-25267,537,-28647,-2529
C04049=4632,34830,-25253,536,-28652,-2533
C04050=4634,34844,-25236,535,-28657,-2534
C04051=4644,34856,-25222,534,-28661,-2537
C04052=4651,34868,-25206,533,-28666,-2540
C04053=4655,34881,-25190,532,-28671,-2542
C04054=4657,34895,-25174,532,-28676,-2542
C04055=4665,34907,-25159,530,-28681,-2545
C04056=4669,34921,-25142,530,-28686,-2547
C04057=4672,34934,-25126,529,-28691,-2548
C04058=4680,34947,-25111,528,-28696,-2551
C04059=4678,34961,-25093,528,-28701,-2550
C04060=4676,34976,-25075,529,-28707,-2549
C04061=4674,34991,-25058,529,-28712,-2549
C04062=4673,35005,-25040,529,-28718,-2548
C04063=4671,35020,-25022,529,-28723,-2547
C04064=4669,35035,-25004,529,-28729,-2546
C04065=4661,35046,-24991,530,-28733,-2543
C04066=4656,35059,-24975,531,-28737,-2541
C04067=4654,35074,-24957,531,-28743,-2540
C04068=4644,35084,-24945,532,-28746,-2536
C04069=4642,35098,-24928,533,-28752,-2535
C04070=4640,35112,-24910,533,-28757,-2535
C04071=4638,35127,-24892,533,-28763,-2534
C04072=4638,35127,-23492,533,-28763,-2534
C04073=5068,35120,-20897,473,-28765,-2702
C04074=5068,35120,-24897,473,-28765,-2702
C04075=5074,35136,-24877,472,-28772,-2705
C04076=5078,35144,-24868,471,-28775,-2706
C04077=5085,35128,-24887,471,-28769,-2709
C04078=5086,35110,-24909,471,-28762,-2709
C04079=5080,35094,-24928,471,-28756,-2707
C04080=5082,35075,-24951,471,-28749,-2708
C04081=5075,35060,-24970,472,-28743,-2705
C04082=5077,35041,-24992,472,-28736,-2706
C04083=5071,35025,-25012,473,-28730,-2704
C04084=5067,35008,-25032,474,-28724,-2702
C04085=5055,34993,-25050,475,-28718,-2698
C04086=5046,34978,-25069,477,-28712,-2694
C04087=5040,34962,-25089,478,-28706,-2692
C04088=5028,34947,-25107,480,-28700,-2687
C04089=5017,34932,-25125,481,-28695,-2683
C04090=5005,34917,-25144,483,-28689,-2678
C04091=4993,34902,-25162,485,-28683,-2674
C04092=4982,34887,-25180,486,-28677,-2670
C04093=4970,34872,-25198,488,-28672,-2665
C04094=4959,34857,-25216,490,-28666,-2661
C04095=4954,34841,-25237,490,-28660,-2659
C04096=4943,34826,-25255,492,-28654,-2654
C04097=4931,34811,-25273,494,-28648,-2650
C04098=4920,34796,-25291,496,-28642,-2645
C04099=4908,34781,-25310,497,-28637,-2641
C04100=4896,34766,-25328,499,-28631,-2637
C04101=4885,34751,-25346,501,-28625,-2632
C04102=4873,34736,-25364,502,-28620,-2628
C04103=4862,34721,-25382,504,-28614,-2623
C04104=4850,34706,-25401,506,-28608,-2619
C04105=4838,34692,-25419,508,-28602,-2614
C04106=4820,34689,-25422,510,-28601,-2607
C04107=4824,34706,-25402,510,-28608,-2608
C04108=4839,34714,-25391,507,-28611,-2614
C04109=4851,34729,-25373,506,-28617,-2619
C04110=4863,34744,-25355,504,-28622,-2623
C04111=4874,34759,-25336,502,-28628,-2628
C04112=4886,34774,-25318,500,-28634,-2632
C04113=4897,34789,-25300,499,-28640,-2637
C04114=4903,34805,-25280,498,-28646,-2639
C04115=4913,34820,-25262,496,-28652,-2643
C04116=4925,34835,-25243,495,-28657,-2647
C04117=4936,34850,-25225,493,-28663,-2652
C04118=4948,34865,-25207,491,-28669,-2656
C04119=4952,34882,-25187,490,-28675,-2658
C04120=4964,34897,-25168,489,-28681,-2662
C04121=4976,34912,-25150,487,-28686,-2667
C04122=4987,34927,-25132,485,-28692,-2671
C04123=4999,34942,-25114,484,-28698,-2676
C04124=5010,34957,-25096,482,-28704,-2680
C04125=5022,34971,-25077,480,-28709,-2685
C04126=5033,34986,-25059,479,-28715,-2689
C04127=5043,35002,-25040,477,-28721,-2693
C04128=5049,35018,-25021,476,-28727,-2695
C04129=5053,35035,-25000,475,-28733,-2697
C04130=5058,35051,-24980,475,-28740,-2699
C04131=5064,35068,-24960,474,-28746,-2701
C04132=5067,35085,-24940,473,-28752,-2702
C04133=5069,35102,-24919,473,-28759,-2703
C04134=5068,35120,-24897,473,-28765,-2702
C04135=5068,35120,-23497,473,-28765,-2702
C04136=5555,35249,-20735,404,-28820,-2893
C04137=5555,35249,-24735,404,-28820,-2893
C04138=5594,35041,-24988,400,-28743,-2909
C04139=5564,34834,-25238,405,-28665,-2898
C04140=5481,34641,-25474,418,-28591,-2866
C04141=5356,34457,-25698,436,-28521,-2817
C04142=5186,34327,-25858,461,-28470,-2751
C04143=4987,34244,-25960,489,-28437,-2674
C04144=4770,34193,-26024,520,-28415,-2589
C04145=4545,34170,-26054,552,-28404,-2501
C04146=4329,34179,-26045,582,-28405,-2417
C04147=4364,34033,-26221,579,-28351,-2431
C04148=4518,33885,-26399,558,-28297,-2492
C04149=4708,33780,-26524,532,-28261,-2567
C04150=4903,33697,-26624,505,-28232,-2644
C04151=5104,33629,-26704,476,-28209,-2722
C04152=5309,33573,-26771,448,-28190,-2802
C04153=5525,33557,-26789,417,-28186,-2887
C04154=5345,33547,-26803,443,-28181,-2817
C04155=5139,33596,-26745,472,-28197,-2736
C04156=4937,33662,-26666,500,-28219,-2657
C04157=4739,33740,-26573,527,-28246,-2579
C04158=4644,33723,-26595,541,-28238,-2542
C04159=4761,33553,-26800,526,-28176,-2589
C04160=4884,33386,-27001,509,-28115,-2638
C04161=5021,33227,-27193,491,-28058,-2692
C04162=5172,33076,-27375,470,-28003,-2751
C04163=5345,32943,-27535,446,-27955,-2819
C04164=5217,33009,-27456,464,-27978,-2769
C04165=5060,33157,-27278,486,-28032,-2707
C04166=4923,33316,-27086,504,-28090,-2653
C04167=4786,33475,-26894,523,-28147,-2599
C04168=4670,33645,-26689,538,-28210,-2553
C04169=4567,33823,-26474,551,-28275,-2512
C04170=4574,33642,-26694,552,-28207,-2515
C04171=4629,33436,-26943,545,-28131,-2538
C04172=4712,33246,-27172,535,-28061,-2571
C04173=4842,33083,-27368,517,-28002,-2622
C04174=5012,32943,-27537,494,-27951,-2689
C04175=5202,32832,-27671,467,-27912,-2764
C04176=5398,32735,-27787,440,-27878,-2840
C04177=5596,32645,-27895,412,-27846,-2918
C04178=5798,32569,-27985,383,-27820,-2997
C04179=5999,32486,-28084,355,-27791,-3075
C04180=6133,32619,-27922,335,-27842,-3127
C04181=6185,32821,-27677,326,-27918,-3146
C04182=6185,33034,-27418,325,-27998,-3146
C04183=6184,33248,-27159,325,-28078,-3145
C04184=6184,33462,-26899,324,-28158,-3144
C04185=6183,33675,-26640,323,-28238,-3143
C04186=6182,33889,-26380,322,-28318,-3142
C04187=6180,34103,-26121,321,-28398,-3141
C04188=6179,34316,-25861,321,-28478,-3140
C04189=6167,34532,-25599,321,-28559,-3134
C04190=6136,34746,-25341,325,-28639,-3122
C04191=6076,34951,-25092,333,-28715,-3098
C04192=5996,35143,-24859,343,-28786,-3066
C04193=5865,35306,-24662,361,-28846,-3014
C04194=5695,35440,-24502,384,-28893,-2947
C04195=5498,35507,-24422,411,-28916,-2870
C04196=5425,35411,-24540,422,-28879,-2841
C04197=5555,35249,-23335,404,-28820,-2893
C04198=-41004,59868,4099,4900,-34257,16705
C04199=-41004,59868,1099,4900,-34257,16705
C04200=-41004,64596,1380,5213,-31659,16463
C04201=-41004,59868,1099,4900,-34257,16705
C04202=-41004,59868,9099,4900,-34257,16705
C04203=5555,35249,-20735,404,-28820,-2893
C04204=5555,35249,-24735,404,-28820,-2893
C04205=5555,35249,-23335,404,-28820,-2893
C04206=6127,35340,-20619,324,-28862,-3117
C04207=6127,35340,-24619,324,-28862,-3117
C04208=6094,35433,-24506,328,-28896,-3103
C04209=6060,35526,-24394,333,-28931,-3090
C04210=6027,35619,-24281,337,-28965,-3077
C04211=6002,35717,-24162,340,-29002,-3067
C04212=5968,35809,-24050,344,-29036,-3053
C04213=5928,35898,-23943,350,-29069,-3037
C04214=5896,35992,-23830,354,-29103,-3024
C04215=5863,36085,-23717,358,-29138,-3011
C04216=5825,36175,-23608,363,-29171,-2996
C04217=5788,36266,-23498,368,-29204,-2982
C04218=5756,36359,-23385,372,-29239,-2969
C04219=5723,36452,-23273,376,-29273,-2955
C04220=5706,36540,-23166,378,-29306,-2948
C04221=5740,36447,-23278,374,-29272,-2962
C04222=5767,36351,-23395,370,-29236,-2973
C04223=5808,36263,-23501,365,-29204,-2989
C04224=5842,36171,-23613,361,-29170,-3003
C04225=5882,36082,-23720,355,-29137,-3019
C04226=5915,35989,-23833,351,-29102,-3032
C04227=5948,35896,-23946,347,-29068,-3045
C04228=5985,35805,-24055,342,-29034,-3060
C04229=6014,35710,-24171,338,-28999,-3071
C04230=6047,35616,-24284,334,-28964,-3085
C04231=6080,35523,-24397,330,-28930,-3098
C04232=6113,35430,-24509,326,-28895,-3111
C04233=6147,35337,-24622,321,-28861,-3124
C04234=6180,35244,-24735,317,-28826,-3138
C04235=6204,35146,-24854,314,-28790,-3147
C04236=6238,35053,-24967,310,-28755,-3161
C04237=6271,34960,-25079,305,-28721,-3174
C04238=6300,34864,-25195,301,-28685,-3186
C04239=6329,34768,-25311,298,-28650,-3197
C04240=6351,34668,-25433,295,-28612,-3206
C04241=6369,34566,-25556,293,-28574,-3213
C04242=6389,34465,-25679,290,-28536,-3221
C04243=6409,34364,-25801,288,-28499,-3229
C04244=6425,34261,-25927,286,-28460,-3236
C04245=6440,34157,-26053,284,-28421,-3242
C04246=6456,34053,-26179,282,-28383,-3248
C04247=6461,33952,-26302,282,-28345,-3251
C04248=6477,33848,-26427,280,-28306,-3257
C04249=6482,33747,-26550,280,-28268,-3259
C04250=6465,33656,-26661,283,-28234,-3253
C04251=6460,33758,-26538,283,-28272,-3251
C04252=6455,33859,-26415,283,-28310,-3249
C04253=6450,33960,-26292,284,-28348,-3246
C04254=6435,34064,-26166,285,-28386,-3240
C04255=6419,34167,-26040,287,-28425,-3234
C04256=6405,34263,-25924,289,-28461,-3228
C04257=6389,34367,-25798,291,-28500,-3222
C04258=6374,34470,-25673,293,-28538,-3215
C04259=6349,34569,-25553,296,-28575,-3205
C04260=6334,34672,-25428,297,-28614,-3199
C04261=6309,34771,-25308,301,-28650,-3189
C04262=6285,34869,-25189,304,-28687,-3179
C04263=6251,34962,-25076,308,-28721,-3166
C04264=6218,35055,-24964,312,-28756,-3153
C04265=6185,35149,-24851,317,-28790,-3140
C04266=6160,35247,-24732,320,-28827,-3130
C04267=6127,35340,-24619,324,-28862,-3117
C04268=6127,35340,-23219,324,-28862,-3117
C04269=6358,35382,-20566,292,-28880,-3207
C04270=6358,35382,-24566,292,-28880,-3207
C04271=6352,35395,-24550,292,-28885,-3205
C04272=6357,35399,-24544,292,-28887,-3206
C04273=6369,35390,-24555,290,-28884,-3211
C04274=6375,35378,-24571,289,-28879,-3214
C04275=6386,35367,-24583,288,-28875,-3218
C04276=6388,35352,-24601,287,-28870,-3219
C04277=6399,35342,-24613,286,-28866,-3223
C04278=6402,35327,-24632,286,-28860,-3224
C04279=6413,35317,-24644,284,-28857,-3229
C04280=6415,35302,-24662,284,-28851,-3230
C04281=6419,35288,-24679,283,-28846,-3231
C04282=6429,35277,-24692,282,-28842,-3235
C04283=6431,35262,-24710,282,-28836,-3236
C04284=6437,35249,-24726,281,-28831,-3238
C04285=6445,35237,-24741,280,-28827,-3241
C04286=6447,35222,-24759,280,-28821,-3242
C04287=6456,35211,-24773,278,-28817,-3246
C04288=6461,35197,-24789,278,-28812,-3248
C04289=6463,35182,-24808,278,-28806,-3249
C04290=6465,35167,-24826,277,-28801,-3250
C04291=6474,35156,-24839,276,-28797,-3253
C04292=6479,35142,-24856,275,-28792,-3255
C04293=6481,35127,-24875,275,-28786,-3256
C04294=6484,35111,-24893,275,-28780,-3257
C04295=6493,35100,-24906,274,-28776,-3260
C04296=6497,35086,-24923,273,-28771,-3262
C04297=6499,35071,-24942,273,-28765,-3263
C04298=6502,35056,-24960,272,-28760,-3264
C04299=6504,35041,-24978,272,-28754,-3265
C04300=6506,35026,-24997,272,-28748,-3266
C04301=6509,35011,-25015,272,-28743,-3267
C04302=6500,35004,-25024,273,-28740,-3263
C04303=6498,35019,-25005,273,-28746,-3262
C04304=6494,35033,-24988,274,-28751,-3261
C04305=6484,35044,-24975,275,-28755,-3257
C04306=6482,35059,-24957,275,-28761,-3256
C04307=6479,35074,-24939,276,-28766,-3255
C04308=6477,35089,-24920,276,-28772,-3254
C04309=6475,35104,-24902,276,-28777,-3253
C04310=6469,35117,-24886,277,-28782,-3251
C04311=6461,35129,-24872,278,-28787,-3248
C04312=6459,35144,-24853,278,-28792,-3247
C04313=6457,35159,-24835,278,-28798,-3246
C04314=6445,35169,-24823,280,-28802,-3242
C04315=6443,35184,-24805,280,-28807,-3241
C04316=6441,35200,-24786,281,-28813,-3240
C04317=6438,35215,-24768,281,-28819,-3239
C04318=6427,35225,-24756,282,-28822,-3234
C04319=6425,35240,-24738,283,-28828,-3234
C04320=6414,35250,-24726,284,-28831,-3229
C04321=6411,35265,-24707,285,-28837,-3228
C04322=6409,35280,-24689,285,-28843,-3227
C04323=6401,35292,-24674,286,-28847,-3224
C04324=6395,35305,-24659,287,-28852,-3222
C04325=6389,35318,-24643,287,-28857,-3219
C04326=6382,35330,-24629,288,-28861,-3217
C04327=6380,35345,-24610,289,-28867,-3216
C04328=6370,35356,-24597,290,-28871,-3212
C04329=6366,35370,-24580,290,-28876,-3210
C04330=6358,35382,-24566,292,-28880,-3207
C04331=6358,35382,-23166,292,-28880,-3207
C04332=5892,34765,-21319,359,-28643,-3026
C04333=5892,34765,-25319,359,-28643,-3026
C04334=5902,34734,-25357,358,-28631,-3030
C04335=5889,34687,-25414,360,-28614,-3025
C04336=5873,34641,-25470,362,-28596,-3019
C04337=5856,34595,-25526,365,-28579,-3012
C04338=5830,34551,-25579,369,-28562,-3003
C04339=5806,34507,-25633,373,-28545,-2993
C04340=5780,34464,-25686,376,-28529,-2983
C04341=5755,34420,-25740,380,-28512,-2973
C04342=5726,34377,-25792,384,-28496,-2962
C04343=5704,34332,-25847,388,-28479,-2954
C04344=5679,34288,-25900,392,-28462,-2944
C04345=5646,34246,-25951,396,-28446,-2932
C04346=5609,34211,-25994,402,-28432,-2917
C04347=5566,34186,-26026,408,-28422,-2901
C04348=5529,34151,-26067,413,-28409,-2886
C04349=5481,34134,-26089,420,-28402,-2868
C04350=5432,34118,-26109,427,-28395,-2849
C04351=5384,34101,-26129,434,-28388,-2830
C04352=5336,34085,-26150,441,-28382,-2811
C04353=5283,34077,-26160,449,-28378,-2790
C04354=5229,34069,-26170,456,-28375,-2769
C04355=5176,34061,-26180,464,-28371,-2748
C04356=5122,34053,-26190,471,-28367,-2728
C04357=5069,34046,-26200,479,-28364,-2707
C04358=5018,34048,-26198,486,-28364,-2687
C04359=4968,34050,-26196,493,-28364,-2667
C04360=4914,34042,-26206,501,-28361,-2646
C04361=4863,34044,-26204,508,-28361,-2627
C04362=4813,34046,-26201,515,-28361,-2607
C04363=4764,34055,-26191,522,-28364,-2588
C04364=4766,34068,-26175,522,-28369,-2588
C04365=4817,34066,-26177,514,-28369,-2608
C04366=4867,34064,-26180,507,-28368,-2628
C04367=4918,34062,-26182,500,-28368,-2648
C04368=4968,34060,-26184,493,-28368,-2668
C04369=5021,34064,-26179,486,-28370,-2688
C04370=5073,34065,-26176,478,-28371,-2708
C04371=5126,34073,-26166,471,-28375,-2729
C04372=5179,34081,-26156,463,-28378,-2750
C04373=5233,34089,-24746,456,-28382,-2771
C04374=-41004,59868,4099,4900,-34257,16705
C04375=-41004,59868,1099,4900,-34257,16705
C04376=-41004,64596,1380,5213,-31659,16463
C04377=-41004,59868,1099,4900,-34257,16705
C04378=-41004,59868,9099,4900,-34257,16705
C04379=5233,34089,-22146,456,-28382,-2771
C04380=5233,34089,-26146,456,-28382,-2771
C04381=5286,34097,-26136,448,-28385,-2792
C04382=5339,34106,-26125,440,-28389,-2812
C04383=5388,34121,-26105,433,-28396,-2831
C04384=5436,34138,-26085,427,-28403,-2850
C04385=5484,34154,-26064,420,-28409,-2869
C04386=5527,34180,-26033,413,-28419,-2885
C04387=5570,34205,-26002,407,-28429,-2902
C04388=5607,34240,-25959,402,-28443,-2916
C04389=5643,34276,-25915,397,-28457,-2930
C04390=5676,34318,-25864,392,-28473,-2943
C04391=5701,34362,-25810,388,-28490,-2953
C04392=5721,34407,-25755,385,-28507,-2961
C04393=5752,34450,-25703,380,-28523,-2972
C04394=5777,34494,-25650,377,-28540,-2982
C04395=5803,34537,-25597,373,-28557,-2992
C04396=5828,34581,-25543,369,-28573,-3002
C04397=5848,34626,-25488,366,-28590,-3009
C04398=5864,34672,-25432,364,-28608,-3015
C04399=5881,34718,-25377,361,-28625,-3022
C04400=5892,34765,-25319,359,-28643,-3026
C04401=5892,34765,-23919,359,-28643,-3026
C04402=5997,34698,-21400,345,-28619,-3067
C04403=5997,34698,-25400,345,-28619,-3067
C04404=6013,34644,-25465,343,-28599,-3074
C04405=6001,34590,-25531,345,-28579,-3069
C04406=5990,34536,-25596,346,-28558,-3065
C04407=5982,34481,-25663,348,-28538,-3062
C04408=5967,34428,-25728,350,-28518,-3056
C04409=5952,34375,-25792,353,-28498,-3051
C04410=5929,34324,-25855,356,-28478,-3042
C04411=5907,34273,-25917,359,-28459,-3033
C04412=5884,34221,-25979,363,-28439,-3025
C04413=5847,34174,-26038,368,-28421,-3010
C04414=5810,34126,-26096,374,-28402,-2996
C04415=5766,34090,-26140,380,-28389,-2979
C04416=5725,34049,-26190,386,-28373,-2963
C04417=5676,34020,-26226,393,-28361,-2944
C04418=5627,33990,-26262,400,-28350,-2925
C04419=5576,33967,-26291,408,-28340,-2905
C04420=5520,33949,-26313,416,-28333,-2883
C04421=5465,33931,-26335,424,-28326,-2862
C04422=5409,33913,-26357,432,-28318,-2840
C04423=5348,33905,-26369,440,-28314,-2816
C04424=5293,33887,-26391,448,-28307,-2795
C04425=5232,33878,-26402,457,-28303,-2771
C04426=5171,33869,-26413,466,-28299,-2747
C04427=5113,33870,-26412,474,-28299,-2725
C04428=5055,33871,-26412,482,-28298,-2702
C04429=4998,33876,-26406,490,-28300,-2680
C04430=4942,33883,-26398,498,-28302,-2658
C04431=4887,33897,-26382,506,-28306,-2636
C04432=4831,33905,-26372,513,-28309,-2615
C04433=4777,33918,-26357,521,-28313,-2593
C04434=4804,33932,-26340,517,-28318,-2604
C04435=4858,33919,-26355,510,-28314,-2625
C04436=4914,33911,-26364,502,-28312,-2647
C04437=4968,33897,-26381,494,-28307,-2668
C04438=5026,33896,-26382,486,-28307,-2691
C04439=5084,33895,-26383,478,-28308,-2713
C04440=5142,33893,-26384,469,-28308,-2736
C04441=5202,33898,-26378,461,-28310,-2759
C04442=5259,33905,-26369,453,-28313,-2782
C04443=5317,33919,-26351,445,-28319,-2804
C04444=5378,33928,-26340,436,-28323,-2828
C04445=5433,33946,-26318,428,-28331,-2849
C04446=5491,33959,-26301,420,-28336,-2872
C04447=5544,33981,-26274,412,-28345,-2893
C04448=5600,33999,-26252,404,-28353,-2914
C04449=5650,34025,-26219,397,-28363,-2934
C04450=5697,34057,-26180,390,-28375,-2952
C04451=5741,34093,-26137,384,-28389,-2969
C04452=5782,34134,-26086,378,-28405,-2985
C04453=5823,34176,-26035,372,-28421,-3001
C04454=5856,34225,-25976,367,-28440,-3014
C04455=5883,34275,-25914,363,-28459,-3024
C04456=5905,34326,-25852,359,-28479,-3033
C04457=5928,34377,-25790,356,-28498,-3041
C04458=5945,34430,-25726,353,-28518,-3048
C04459=5958,34484,-25661,351,-28538,-3053
C04460=5973,34537,-25596,349,-28558,-3058
C04461=5981,34591,-25530,347,-28579,-3062
C04462=5993,34645,-25464,346,-28599,-3066
C04463=5997,34698,-25400,345,-28619,-3067
C04464=5997,34698,-24000,345,-28619,-3067
C04465=5383,34790,-21294,431,-28646,-2827
C04466=5383,34790,-25294,431,-28646,-2827
C04467=5368,34766,-25323,433,-28637,-2821
C04468=5361,34740,-25355,434,-28627,-2819
C04469=5345,34717,-25383,436,-28618,-2812
C04470=5338,34691,-25414,437,-28608,-2810
C04471=5322,34668,-25443,440,-28600,-2804
C04472=5312,34643,-25473,441,-28590,-2800
C04473=5301,34618,-25503,443,-28581,-2795
C04474=5283,34595,-25532,446,-28572,-2789
C04475=5273,34570,-25562,447,-28562,-2784
C04476=5255,34547,-25590,450,-28554,-2778
C04477=5237,34524,-25618,453,-28545,-2771
C04478=5215,34507,-25639,456,-28538,-2762
C04479=5197,34484,-25667,458,-28529,-2755
C04480=5176,34467,-25687,461,-28523,-2747
C04481=5154,34451,-25708,465,-28516,-2739
C04482=5135,34429,-25734,467,-28508,-2731
C04483=5111,34416,-25750,471,-28503,-2722
C04484=5089,34400,-25770,474,-28497,-2713
C04485=5064,34390,-25783,478,-28492,-2703
C04486=5042,34373,-25803,481,-28486,-2695
C04487=5017,34362,-25816,484,-28482,-2685
C04488=4995,34345,-25837,488,-28475,-2677
C04489=4970,34335,-25850,491,-28471,-2667
C04490=4948,34318,-25871,494,-28464,-2658
C04491=4923,34307,-25884,498,-28460,-2649
C04492=4897,34297,-25897,502,-28456,-2639
C04493=4873,34285,-25912,505,-28451,-2629
C04494=4849,34272,-25928,509,-28446,-2620
C04495=4825,34259,-25944,512,-28441,-2610
C04496=4838,34280,-25918,510,-28449,-2615
C04497=4862,34293,-25902,507,-28454,-2625
C04498=4886,34305,-25887,503,-28458,-2634
C04499=4912,34315,-25874,500,-28463,-2644
C04500=4937,34326,-25861,496,-28467,-2654
C04501=4959,34343,-25841,493,-28474,-2663
C04502=4981,34358,-25821,489,-28480,-2671
C04503=5006,34370,-25807,486,-28484,-2681
C04504=5029,34384,-25789,483,-28490,-2690
C04505=5053,34398,-25773,479,-28495,-2699
C04506=5077,34411,-25757,476,-28500,-2708
C04507=5096,34431,-25732,473,-28508,-2716
C04508=5119,34446,-25714,470,-28514,-2725
C04509=5143,34459,-25698,466,-28519,-2734
C04510=5162,34481,-25671,463,-28528,-2741
C04511=5183,34498,-25650,460,-28535,-2750
C04512=5201,34521,-25621,458,-28543,-2756
C04513=5218,34545,-25593,455,-28552,-2763
C04514=5236,34568,-25565,452,-28561,-2770
C04515=5254,34591,-25537,450,-28570,-2777
C04516=5272,34614,-25509,447,-28579,-2784
C04517=5283,34638,-25479,446,-28588,-2788
C04518=5301,34661,-25451,443,-28597,-2795
C04519=5311,34686,-25420,441,-28606,-2799
C04520=5322,34711,-25390,440,-28616,-2803
C04521=5333,34736,-25360,438,-28625,-2807
C04522=5349,34759,-25332,436,-28634,-2814
C04523=5355,34785,-25300,435,-28644,-2816
C04524=5372,34808,-25272,432,-28653,-2822
C04525=5388,34814,-25265,430,-28655,-2829
C04526=5383,34790,-25294,431,-28646,-2827
C04527=5383,34790,-23894,431,-28646,-2827
C04528=5143,34689,-21419,465,-28605,-2733
C04529=5143,34689,-25419,465,-28605,-2733
C04530=5130,34668,-25445,467,-28597,-2729
C04531=5111,34648,-25469,470,-28590,-2721
C04532=5090,34632,-25489,473,-28583,-2713
C04533=5069,34616,-25508,476,-28577,-2705
C04534=5048,34599,-25528,479,-28571,-2696
C04535=5026,34585,-25546,482,-28565,-2688
C04536=5002,34572,-25562,485,-28560,-2679
C04537=4981,34557,-25581,488,-28554,-2670
C04538=4960,34541,-25601,491,-28548,-2662
C04539=4938,34524,-25620,495,-28541,-2654
C04540=4914,34514,-25633,498,-28537,-2644
C04541=4892,34498,-25652,501,-28531,-2636
C04542=4867,34488,-25665,505,-28527,-2626
C04543=4846,34472,-25684,508,-28521,-2618
C04544=4821,34462,-25697,511,-28516,-2608
C04545=4799,34446,-25716,515,-28510,-2600
C04546=4775,34435,-25730,518,-28506,-2590
C04547=4750,34425,-25742,522,-28502,-2581
C04548=4725,34415,-25755,525,-28498,-2571
C04549=4702,34403,-24369,529,-28493,-2562
C04550=-41004,59868,4099,4900,-34257,16705
C04551=-41004,59868,1099,4900,-34257,16705
C04552=-41004,64596,1380,5213,-31659,16463
C04553=-41004,59868,1099,4900,-34257,16705
C04554=-41004,59868,9099,4900,-34257,16705
C04555=4702,34403,-21769,529,-28493,-2562
C04556=4702,34403,-25769,529,-28493,-2562
C04557=4678,34390,-25785,532,-28488,-2553
C04558=4651,34385,-25792,536,-28486,-2542
C04559=4627,34373,-25807,539,-28481,-2533
C04560=4604,34360,-25823,543,-28476,-2524
C04561=4576,34355,-25829,547,-28474,-2513
C04562=4552,34343,-25844,550,-28469,-2504
C04563=4529,34330,-25860,553,-28464,-2494
C04564=4500,34326,-25865,557,-28462,-2483
C04565=4472,34322,-25871,561,-28460,-2472
C04566=4444,34318,-25876,565,-28458,-2461
C04567=4461,34330,-25861,563,-28463,-2468
C04568=4490,34334,-25856,559,-28465,-2479
C04569=4513,34347,-25840,555,-28470,-2488
C04570=4541,34351,-25834,551,-28472,-2499
C04571=4565,34363,-25819,548,-28476,-2508
C04572=4590,34373,-25807,544,-28481,-2518
C04573=4616,34381,-25797,541,-28484,-2528
C04574=4640,34393,-25782,537,-28489,-2538
C04575=4665,34403,-25770,534,-28493,-2547
C04576=4691,34411,-25760,530,-28496,-2557
C04577=4714,34424,-25744,527,-28501,-2567
C04578=4737,34437,-25728,523,-28506,-2576
C04579=4761,34450,-25713,520,-28511,-2585
C04580=4786,34460,-25700,516,-28515,-2594
C04581=4807,34476,-25680,513,-28522,-2603
C04582=4830,34489,-25664,510,-28527,-2612
C04583=4853,34502,-25648,507,-28532,-2621
C04584=4876,34515,-25632,503,-28537,-2630
C04585=4899,34528,-25616,500,-28542,-2639
C04586=4922,34541,-25600,497,-28547,-2648
C04587=4945,34554,-25584,493,-28552,-2657
C04588=4969,34567,-25568,490,-28558,-2666
C04589=4991,34581,-25551,487,-28563,-2674
C04590=5012,34597,-25531,484,-28569,-2682
C04591=5033,34614,-25511,481,-28576,-2691
C04592=5055,34630,-25491,478,-28582,-2699
C04593=5076,34646,-25471,475,-28588,-2707
C04594=5097,34662,-25452,471,-28595,-2715
C04595=5118,34679,-25432,468,-28601,-2724
C04596=5143,34689,-25419,465,-28605,-2733
C04597=5143,34689,-24019,465,-28605,-2733
C04598=5124,34510,-21636,469,-28538,-2726
C04599=5124,34510,-25636,469,-28538,-2726
C04600=5111,34494,-25656,470,-28532,-2721
C04601=5094,34483,-25669,473,-28528,-2715
C04602=5078,34473,-25681,475,-28524,-2709
C04603=5061,34463,-25694,478,-28520,-2702
C04604=5044,34454,-25705,480,-28516,-2695
C04605=5028,34442,-25719,482,-28512,-2689
C04606=5008,34438,-25725,485,-28510,-2681
C04607=4991,34427,-25738,488,-28505,-2675
C04608=4971,34424,-25742,491,-28504,-2667
C04609=4955,34412,-25757,493,-28499,-2661
C04610=4938,34403,-25768,495,-28496,-2654
C04611=4918,34397,-25775,498,-28493,-2647
C04612=4901,34389,-25786,501,-28490,-2640
C04613=4882,34382,-25794,503,-28487,-2632
C04614=4861,34379,-25798,506,-28486,-2624
C04615=4845,34367,-25812,509,-28481,-2618
C04616=4824,34364,-25816,512,-28480,-2610
C04617=4809,34352,-25831,514,-28475,-2604
C04618=4788,34349,-25835,517,-28474,-2596
C04619=4770,34341,-25844,519,-28471,-2589
C04620=4751,34334,-25853,522,-28468,-2581
C04621=4730,34331,-25857,525,-28466,-2573
C04622=4709,34328,-25861,528,-28465,-2565
C04623=4694,34316,-25875,530,-28460,-2559
C04624=4673,34313,-25879,533,-28459,-2551
C04625=4652,34310,-25883,536,-28458,-2543
C04626=4631,34307,-25887,539,-28456,-2534
C04627=4615,34296,-25901,541,-28452,-2528
C04628=4594,34292,-25906,544,-28450,-2520
C04629=4602,34295,-25902,543,-28451,-2523
C04630=4619,34302,-25894,541,-28454,-2530
C04631=4627,34316,-25876,540,-28460,-2533
C04632=4648,34319,-25872,537,-28461,-2541
C04633=4669,34322,-25868,534,-28462,-2549
C04634=4689,34326,-25863,531,-28464,-2557
C04635=4706,34337,-25850,528,-28468,-2564
C04636=4727,34340,-25846,525,-28470,-2572
C04637=4747,34345,-25840,523,-28472,-2580
C04638=4763,34355,-25828,520,-28476,-2586
C04639=4784,34359,-25822,517,-28478,-2594
C04640=4800,34370,-25809,515,-28482,-2600
C04641=4820,34373,-25805,512,-28483,-2608
C04642=4836,34385,-25791,510,-28488,-2615
C04643=4857,34388,-25787,507,-28489,-2623
C04644=4874,34398,-25774,504,-28493,-2629
C04645=4894,34403,-25768,502,-28495,-2637
C04646=4911,34413,-25756,499,-28499,-2644
C04647=4930,34418,-25750,496,-28501,-2651
C04648=4948,34427,-25738,494,-28505,-2658
C04649=4967,34433,-25731,491,-28507,-2665
C04650=4985,34441,-25721,489,-28511,-2672
C04651=5004,34448,-25713,486,-28513,-2680
C04652=5021,34456,-25703,483,-28517,-2687
C04653=5040,34463,-25694,481,-28519,-2694
C04654=5055,34473,-25682,478,-28523,-2700
C04655=5074,34468,-25688,476,-28522,-2707
C04656=5089,34480,-25673,474,-28526,-2713
C04657=5099,34496,-25654,472,-28533,-2717
C04658=5115,34503,-25645,470,-28535,-2723
C04659=5124,34510,-25636,469,-28538,-2726
C04660=5124,34510,-24236,469,-28538,-2726
C04661=4468,34663,-21457,560,-28587,-2469
C04662=4468,34663,-25457,560,-28587,-2469
C04663=4461,34654,-25468,561,-28584,-2466
C04664=4454,34645,-25479,562,-28580,-2464
C04665=4447,34636,-25490,563,-28577,-2461
C04666=4440,34627,-25501,564,-28573,-2458
C04667=4432,34618,-25512,565,-28570,-2455
C04668=4429,34608,-25524,566,-28566,-2454
C04669=4425,34598,-25536,566,-28562,-2453
C04670=4418,34589,-25548,567,-28559,-2450
C04671=4411,34580,-25559,568,-28555,-2447
C04672=4404,34570,-25570,569,-28552,-2445
C04673=4397,34561,-25581,570,-28548,-2442
C04674=4390,34552,-25592,571,-28545,-2439
C04675=4382,34543,-25603,572,-28541,-2436
C04676=4375,34534,-25614,574,-28538,-2433
C04677=4368,34525,-25625,575,-28534,-2431
C04678=4361,34516,-25636,576,-28531,-2428
C04679=4354,34507,-25648,577,-28527,-2425
C04680=4354,34496,-25661,577,-28523,-2425
C04681=4347,34487,-25672,578,-28520,-2422
C04682=4340,34478,-25683,579,-28516,-2420
C04683=4332,34468,-25694,580,-28513,-2417
C04684=4325,34459,-25705,581,-28509,-2414
C04685=4318,34450,-25716,582,-28506,-2411
C04686=4311,34441,-25727,583,-28502,-2409
C04687=4304,34432,-25738,584,-28499,-2406
C04688=4293,34429,-25742,586,-28498,-2402
C04689=4286,34420,-25753,587,-28494,-2399
C04690=4275,34417,-25757,588,-28493,-2395
C04691=4286,34420,-25753,587,-28494,-2399
C04692=4293,34429,-25742,586,-28498,-2402
C04693=4293,34440,-25729,586,-28502,-2402
C04694=4300,34449,-25718,585,-28505,-2404
C04695=4307,34458,-25707,584,-28509,-2407
C04696=4314,34467,-25696,583,-28512,-2410
C04697=4317,34478,-25683,582,-28516,-2411
C04698=4322,34487,-25671,581,-28520,-2413
C04699=4329,34496,-25660,580,-28523,-2415
C04700=4336,34506,-25649,579,-28527,-2418
C04701=4343,34515,-25638,578,-28530,-2421
C04702=4350,34524,-25627,577,-28534,-2424
C04703=4350,34535,-25614,577,-28538,-2424
C04704=4357,34544,-25603,576,-28541,-2426
C04705=4365,34553,-25591,575,-28545,-2429
C04706=4372,34562,-25580,574,-28548,-2432
C04707=4379,34571,-25569,573,-28552,-2435
C04708=4386,34580,-25558,572,-28555,-2437
C04709=4393,34589,-25547,571,-28559,-2440
C04710=4400,34598,-25536,570,-28562,-2443
C04711=4407,34608,-25525,569,-28566,-2446
C04712=4408,34618,-25512,568,-28570,-2446
C04713=4415,34627,-25500,567,-28573,-2448
C04714=4422,34637,-25489,566,-28577,-2451
C04715=4429,34646,-25478,565,-28580,-2454
C04716=4436,34655,-25467,564,-28584,-2457
C04717=4443,34664,-25456,563,-28587,-2459
C04718=4450,34673,-25445,562,-28591,-2462
C04719=4457,34682,-25434,561,-28594,-2465
C04720=4468,34685,-25430,560,-28595,-2469
C04721=4469,34674,-25444,559,-28591,-2470
C04722=4468,34663,-24057,560,-28587,-2469
C04723=-41004,59868,4099,4900,-34257,16705
C04724=-41004,59868,1099,4900,-34257,16705
C04725=-41004,64596,1380,5213,-31659,16463
C04726=-41004,59868,1099,4900,-34257,16705
C04727=-41004,59868,9099,4900,-34257,16705
C04728=4468,34663,-21457,560,-28587,-2469
C04729=4468,34663,-25457,560,-28587,-2469
C04730=4468,34663,-24057,560,-28587,-2469
C04731=3987,34709,-21406,627,-28598,-2281
C04732=3987,34709,-25406,627,-28598,-2281
C04733=3980,34685,-25435,628,-28589,-2278
C04734=3974,34661,-25464,629,-28580,-2276
C04735=3976,34635,-25495,629,-28571,-2277
C04736=3969,34612,-25524,630,-28562,-2274
C04737=3967,34587,-25554,630,-28552,-2273
C04738=3957,34564,-25582,632,-28544,-2270
C04739=3947,34541,-25610,633,-28535,-2266
C04740=3937,34518,-25638,635,-28526,-2262
C04741=3923,34496,-25665,637,-28518,-2257
C04742=3911,34473,-25692,639,-28509,-2252
C04743=3901,34450,-25721,641,-28501,-2248
C04744=3884,34429,-25747,643,-28492,-2242
C04745=3874,34406,-25775,645,-28484,-2238
C04746=3858,34384,-25801,647,-28476,-2232
C04747=3841,34363,-25827,650,-28467,-2225
C04748=3820,34348,-25845,653,-28462,-2217
C04749=3803,34327,-25871,655,-28453,-2211
